LIN {X 0,Y 131.73,Z 570.995,A -85,B 0,C 180,E1 -25686.554,E2 -25686.554} C_VEL
LIN {X 0,Y 133.892,Z 570.97,A -85,B 0,C 180,E1 -25688.915,E2 -25688.915} C_VEL
LIN {X 0,Y 134.91,Z 571.003,A -85,B 0,C 180,E1 -25689.63,E2 -25689.63} C_VEL
LIN {X 0,Y 142.32,Z 571.103,A -85,B 0,C 180,E1 -25693.736,E2 -25693.736} C_VEL
LIN {X 0,Y 151.999,Z 570.353,A -85,B 0,C 180,E1 -25697.713,E2 -25697.713} C_VEL
LIN {X 0,Y 158.478,Z 569.41,A -85,B 0,C 180,E1 -25699.824,E2 -25699.824} C_VEL
LIN {X 0,Y 159.217,Z 569.07,A -85,B 0,C 180,E1 -25700.5,E2 -25700.5} C_VEL
LIN {X 0,Y 151.909,Z 567.926,A -85,B 0,C 180,E1 -25703.025,E2 -25703.025} C_VEL
LIN {X 0,Y 142.456,Z 565.139,A -85,B 0,C 180,E1 -25707.132,E2 -25707.132} C_VEL
LIN {X 0,Y 134.098,Z 561.047,A -85,B 0,C 180,E1 -25711.855,E2 -25711.855} C_VEL
LIN {X 0,Y 127.082,Z 555.595,A -85,B 0,C 180,E1 -25717.223,E2 -25717.223} C_VEL
LIN {X 0,Y 121.684,Z 548.605,A -85,B 0,C 180,E1 -25723.213,E2 -25723.213} C_VEL
LIN {X 0,Y 117.883,Z 539.949,A -85,B 0,C 180,E1 -25729.695,E2 -25729.695} C_VEL
LIN {X 0,Y 115.994,Z 530.669,A -85,B 0,C 180,E1 -25735.655,E2 -25735.655} C_VEL
LIN {X 0,Y 115.384,Z 519.452,A -85,B 0,C 180,E1 -25741.744,E2 -25741.744} C_VEL
LIN {X 0,Y 115.582,Z 508.598,A -85,B 0,C 180,E1 -25746.545,E2 -25746.545} C_VEL
LIN {X 0,Y 116.083,Z 497.899,A -85,B 0,C 180,E1 -25750.463,E2 -25750.463} C_VEL
LIN {X 0,Y 116.869,Z 485.455,A -85,B 0,C 180,E1 -25754.183,E2 -25754.183} C_VEL
LIN {X 0,Y 117.808,Z 470.89,A -85,B 0,C 180,E1 -25757.577,E2 -25757.577} C_VEL
LIN {X 0,Y 118.72,Z 456.9,A -85,B 0,C 180,E1 -25760.012,E2 -25760.012} C_VEL
LIN {X 0,Y 119.766,Z 433.179,A -85,B 0,C 180,E1 -25762.99,E2 -25762.99} C_VEL
LIN {X 0,Y 121.096,Z 391.719,A -85,B 0,C 180,E1 -25767.775,E2 -25767.775} C_VEL
LIN {X 0,Y 115.765,Z 370.385,A -85,B 0,C 180,E1 -25770.236,E2 -25770.236} C_VEL
LIN {X 0,Y 115.16,Z 367.133,A -85,B 0,C 180,E1 -25770.68,E2 -25770.68} C_VEL
LIN {X 0,Y 114.785,Z 367.181,A -85,B 0,C 180,E1 -25777.752,E2 -25777.752} C_VEL
LIN {X 0,Y 114.785,Z 367.188,A -85,B 0,C 180,E1 -25782.716,E2 -25782.716} C_VEL
LIN {X 0,Y 114.8,Z 367.179,A -85,B 0,C 180,E1 -25787.669,E2 -25787.669} C_VEL
LIN {X 0,Y 114.81,Z 367.183,A -85,B 0,C 180,E1 -25792.727,E2 -25792.727} C_VEL
LIN {X 0,Y 114.866,Z 367.177,A -85,B 0,C 180,E1 -25798.931,E2 -25798.931} C_VEL
LIN {X 0,Y 114.944,Z 367.165,A -85,B 0,C 180,E1 -25806.507,E2 -25806.507} C_VEL
LIN {X 0,Y 115.016,Z 367.152,A -85,B 0,C 180,E1 -25812.211,E2 -25812.211} C_VEL
LIN {X 0,Y 115.284,Z 367.124,A -85,B 0,C 180,E1 -25817.258,E2 -25817.258} C_VEL
LIN {X 0,Y 115.391,Z 367.108,A -85,B 0,C 180,E1 -25819.472,E2 -25819.472} C_VEL
LIN {X 0,Y 115.535,Z 367.093,A -85,B 0,C 180,E1 -25826.513,E2 -25826.513} C_VEL
LIN {X 0,Y 115.994,Z 367.029,A -85,B 0,C 180,E1 -25830.001,E2 -25830.001} C_VEL
LIN {X 0,Y 115.396,Z 367.106,A -85,B 0,C 180,E1 -25836.997,E2 -25836.997} C_VEL
LIN {X 0,Y 115.391,Z 367.109,A -85,B 0,C 180,E1 -25840.529,E2 -25840.529} C_VEL
LIN {X 0,Y 115.146,Z 367.141,A -85,B 0,C 180,E1 -25844.132,E2 -25844.132} C_VEL
LIN {X 0,Y 114.98,Z 367.162,A -85,B 0,C 180,E1 -25851.516,E2 -25851.516} C_VEL
LIN {X 0,Y 114.872,Z 367.169,A -85,B 0,C 180,E1 -25855.359,E2 -25855.359} C_VEL
LIN {X 0,Y 114.867,Z 367.175,A -85,B 0,C 180,E1 -25861.07,E2 -25861.07} C_VEL
LIN {X 0,Y 114.801,Z 367.185,A -85,B 0,C 180,E1 -25867.749,E2 -25867.749} C_VEL
LIN {X 0,Y 114.793,Z 367.179,A -85,B 0,C 180,E1 -25872.723,E2 -25872.723} C_VEL
LIN {X 0,Y 115,Z 367.154,A -85,B 0,C 180,E1 -25880.133,E2 -25880.133} C_VEL
LIN {X 0,Y 122.575,Z 395.545,A -85,B 0,C 180,E1 -25883.546,E2 -25883.546} C_VEL
LIN {X 0,Y 119.952,Z 450.842,A -85,B 0,C 180,E1 -25889.405,E2 -25889.405} C_VEL
LIN {X 0,Y 118.922,Z 465.573,A -85,B 0,C 180,E1 -25891.547,E2 -25891.547} C_VEL
LIN {X 0,Y 117.737,Z 479.37,A -85,B 0,C 180,E1 -25894.314,E2 -25894.314} C_VEL
LIN {X 0,Y 116.517,Z 492.918,A -85,B 0,C 180,E1 -25897.855,E2 -25897.855} C_VEL
LIN {X 0,Y 115.452,Z 506.149,A -85,B 0,C 180,E1 -25902.282,E2 -25902.282} C_VEL
LIN {X 0,Y 114.783,Z 517.895,A -85,B 0,C 180,E1 -25907.313,E2 -25907.313} C_VEL
LIN {X 0,Y 114.688,Z 527.291,A -85,B 0,C 180,E1 -25912.188,E2 -25912.188} C_VEL
LIN {X 0,Y 115.328,Z 535.667,A -85,B 0,C 180,E1 -25917.382,E2 -25917.382} C_VEL
LIN {X 0,Y 117.114,Z 543.83,A -85,B 0,C 180,E1 -25923.442,E2 -25923.442} C_VEL
LIN {X 0,Y 119.746,Z 549.675,A -85,B 0,C 180,E1 -25928.439,E2 -25928.439} C_VEL
LIN {X 0,Y 124.689,Z 555.877,A -85,B 0,C 180,E1 -25934.695,E2 -25934.695} C_VEL
LIN {X 0,Y 129.437,Z 559.537,A -85,B 0,C 180,E1 -25939.014,E2 -25939.014} C_VEL
LIN {X 0,Y 137.108,Z 563.055,A -85,B 0,C 180,E1 -25944.211,E2 -25944.211} C_VEL
LIN {X 0,Y 145.877,Z 565.201,A -85,B 0,C 180,E1 -25948.803,E2 -25948.803} C_VEL
LIN {X 0,Y 150.702,Z 565.75,A -85,B 0,C 180,E1 -25950.864,E2 -25950.864} C_VEL
LIN {X 0,Y 161.056,Z 565.721,A -85,B 0,C 180,E1 -25954.562,E2 -25954.562} C_VEL
LIN {X 0,Y 168.992,Z 564.854,A -85,B 0,C 180,E1 -25956.918,E2 -25956.918} C_VEL
LIN {X 0,Y 168.367,Z 565.266,A -85,B 0,C 180,E1 -25957.522,E2 -25957.522} C_VEL
LIN {X 0,Y 157.071,Z 568.845,A -85,B 0,C 180,E1 -25960.477,E2 -25960.477} C_VEL
LIN {X 0,Y 146.884,Z 571.301,A -85,B 0,C 180,E1 -25964.133,E2 -25964.133} C_VEL
LIN {X 0,Y 137.625,Z 572.661,A -85,B 0,C 180,E1 -25968.404,E2 -25968.404} C_VEL
LIN {X 0,Y 129.744,Z 572.964,A -85,B 0,C 180,E1 -25973.426,E2 -25973.426} C_VEL
LIN {X 0,Y 123.542,Z 572.25,A -85,B 0,C 180,E1 -25979.203,E2 -25979.203} C_VEL
LIN {X 0,Y 119.301,Z 570.519,A -85,B 0,C 180,E1 -25985.645,E2 -25985.645} C_VEL
LIN {X 0,Y 117.086,Z 567.075,A -85,B 0,C 180,E1 -25993.825,E2 -25993.825} C_VEL
LIN {X 0,Y 117.795,Z 562.438,A -85,B 0,C 180,E1 -26001.421,E2 -26001.421} C_VEL
LIN {X 0,Y 119.686,Z 558.145,A -85,B 0,C 180,E1 -26006.633,E2 -26006.633} C_VEL
LIN {X 0,Y 121.553,Z 553.452,A -85,B 0,C 180,E1 -26010.862,E2 -26010.862} C_VEL
LIN {X 0,Y 122.427,Z 551.524,A -85,B 0,C 180,E1 -26012.403,E2 -26012.403} C_VEL
LIN {X 0,Y 119.958,Z 557.118,A -85,B 0,C 180,E1 -26018.252,E2 -26018.252} C_VEL
LIN {X 0,Y 118.732,Z 562.143,A -85,B 0,C 180,E1 -26025.448,E2 -26025.448} C_VEL
LIN {X 0,Y 119.345,Z 565.021,A -85,B 0,C 180,E1 -26030.691,E2 -26030.691} C_VEL
LIN {X 0,Y 122.151,Z 567.945,A -85,B 0,C 180,E1 -26037.405,E2 -26037.405} C_VEL
LIN {X 0,Y 127.121,Z 569.905,A -85,B 0,C 180,E1 -26043.563,E2 -26043.563} C_VEL
LIN {X 0,Y 134.91,Z 571.003,A -85,B 0,C 180,E1 -26049.63,E2 -26049.63} C_VEL
LIN {X 0,Y 136.633,Z 570.98,A -85,B 0,C 180,E1 -26051.153,E2 -26051.153} C_VEL
LIN {X 0,Y 140.12,Z 569.71,A -85,B 0,C 180,E1 -26056.537,E2 -26056.537} C_VEL
LIN {X 0,Y 142.388,Z 569.441,A -85,B 0,C 180,E1 -26057.855,E2 -26057.855} C_VEL
LIN {X 0,Y 148.167,Z 569.104,A -85,B 0,C 180,E1 -26059.993,E2 -26059.993} C_VEL
LIN {X 0,Y 147.74,Z 568.702,A -85,B 0,C 180,E1 -26060.827,E2 -26060.827} C_VEL
LIN {X 0,Y 141.273,Z 566.851,A -85,B 0,C 180,E1 -26063.345,E2 -26063.345} C_VEL
LIN {X 0,Y 132.011,Z 562.872,A -85,B 0,C 180,E1 -26067.832,E2 -26067.832} C_VEL
LIN {X 0,Y 124.058,Z 557.572,A -85,B 0,C 180,E1 -26073.049,E2 -26073.049} C_VEL
LIN {X 0,Y 117.628,Z 550.855,A -85,B 0,C 180,E1 -26078.991,E2 -26078.991} C_VEL
LIN {X 0,Y 112.873,Z 542.487,A -85,B 0,C 180,E1 -26085.576,E2 -26085.576} C_VEL
LIN {X 0,Y 110.207,Z 533.661,A -85,B 0,C 180,E1 -26091.749,E2 -26091.749} C_VEL
LIN {X 0,Y 108.789,Z 522.89,A -85,B 0,C 180,E1 -26098.147,E2 -26098.147} C_VEL
LIN {X 0,Y 108.708,Z 512.813,A -85,B 0,C 180,E1 -26103.241,E2 -26103.241} C_VEL
LIN {X 0,Y 109.057,Z 501.757,A -85,B 0,C 180,E1 -26107.869,E2 -26107.869} C_VEL
LIN {X 0,Y 109.628,Z 489.445,A -85,B 0,C 180,E1 -26112.024,E2 -26112.024} C_VEL
LIN {X 0,Y 110.337,Z 478.245,A -85,B 0,C 180,E1 -26115.101,E2 -26115.101} C_VEL
LIN {X 0,Y 111.269,Z 464.295,A -85,B 0,C 180,E1 -26118.108,E2 -26118.108} C_VEL
LIN {X 0,Y 112.021,Z 449.968,A -85,B 0,C 180,E1 -26120.387,E2 -26120.387} C_VEL
LIN {X 0,Y 112.84,Z 428.51,A -85,B 0,C 180,E1 -26123.149,E2 -26123.149} C_VEL
LIN {X 0,Y 113.972,Z 392.449,A -85,B 0,C 180,E1 -26127.612,E2 -26127.612} C_VEL
LIN {X 0,Y 108.815,Z 371.696,A -85,B 0,C 180,E1 -26130.125,E2 -26130.125} C_VEL
LIN {X 0,Y 108.119,Z 368.01,A -85,B 0,C 180,E1 -26130.619,E2 -26130.619} C_VEL
LIN {X 0,Y 107.691,Z 368.063,A -85,B 0,C 180,E1 -26138.453,E2 -26138.453} C_VEL
LIN {X 0,Y 107.679,Z 368.068,A -85,B 0,C 180,E1 -26145.883,E2 -26145.883} C_VEL
LIN {X 0,Y 107.705,Z 368.068,A -85,B 0,C 180,E1 -26151.536,E2 -26151.536} C_VEL
LIN {X 0,Y 107.804,Z 368.055,A -85,B 0,C 180,E1 -26158.565,E2 -26158.565} C_VEL
LIN {X 0,Y 107.908,Z 368.043,A -85,B 0,C 180,E1 -26166.998,E2 -26166.998} C_VEL
LIN {X 0,Y 108.037,Z 368.026,A -85,B 0,C 180,E1 -26174.918,E2 -26174.918} C_VEL
LIN {X 0,Y 108.304,Z 367.992,A -85,B 0,C 180,E1 -26178.775,E2 -26178.775} C_VEL
LIN {X 0,Y 108.461,Z 367.975,A -85,B 0,C 180,E1 -26186.285,E2 -26186.285} C_VEL
LIN {X 0,Y 108.945,Z 367.907,A -85,B 0,C 180,E1 -26190.001,E2 -26190.001} C_VEL
LIN {X 0,Y 108.338,Z 367.985,A -85,B 0,C 180,E1 -26197.455,E2 -26197.455} C_VEL
LIN {X 0,Y 108.201,Z 368.007,A -85,B 0,C 180,E1 -26203.027,E2 -26203.027} C_VEL
LIN {X 0,Y 107.907,Z 368.042,A -85,B 0,C 180,E1 -26209.006,E2 -26209.006} C_VEL
LIN {X 0,Y 107.857,Z 368.045,A -85,B 0,C 180,E1 -26214.187,E2 -26214.187} C_VEL
LIN {X 0,Y 107.793,Z 368.055,A -85,B 0,C 180,E1 -26222.053,E2 -26222.053} C_VEL
LIN {X 0,Y 107.707,Z 368.069,A -85,B 0,C 180,E1 -26228.465,E2 -26228.465} C_VEL
LIN {X 0,Y 107.7,Z 368.069,A -85,B 0,C 180,E1 -26235.875,E2 -26235.875} C_VEL
LIN {X 0,Y 107.921,Z 368.037,A -85,B 0,C 180,E1 -26239.801,E2 -26239.801} C_VEL
LIN {X 0,Y 115.442,Z 397.023,A -85,B 0,C 180,E1 -26243.484,E2 -26243.484} C_VEL
LIN {X 0,Y 112.956,Z 448.955,A -85,B 0,C 180,E1 -26249.377,E2 -26249.377} C_VEL
LIN {X 0,Y 112.103,Z 462.355,A -85,B 0,C 180,E1 -26251.276,E2 -26251.276} C_VEL
LIN {X 0,Y 110.854,Z 476.95,A -85,B 0,C 180,E1 -26254.162,E2 -26254.162} C_VEL
LIN {X 0,Y 109.706,Z 489.289,A -85,B 0,C 180,E1 -26257.397,E2 -26257.397} C_VEL
LIN {X 0,Y 108.696,Z 502.041,A -85,B 0,C 180,E1 -26261.629,E2 -26261.629} C_VEL
LIN {X 0,Y 108.018,Z 513.424,A -85,B 0,C 180,E1 -26266.361,E2 -26266.361} C_VEL
LIN {X 0,Y 107.775,Z 524.013,A -85,B 0,C 180,E1 -26271.723,E2 -26271.723} C_VEL
LIN {X 0,Y 108.37,Z 532.92,A -85,B 0,C 180,E1 -26277.214,E2 -26277.214} C_VEL
LIN {X 0,Y 110.105,Z 541.774,A -85,B 0,C 180,E1 -26283.661,E2 -26283.661} C_VEL
LIN {X 0,Y 112.721,Z 548.038,A -85,B 0,C 180,E1 -26288.969,E2 -26288.969} C_VEL
LIN {X 0,Y 116.359,Z 553.32,A -85,B 0,C 180,E1 -26293.982,E2 -26293.982} C_VEL
LIN {X 0,Y 120.926,Z 557.672,A -85,B 0,C 180,E1 -26298.643,E2 -26298.643} C_VEL
LIN {X 0,Y 126.435,Z 561.187,A -85,B 0,C 180,E1 -26302.9,E2 -26302.9} C_VEL
LIN {X 0,Y 134.957,Z 564.601,A -85,B 0,C 180,E1 -26307.95,E2 -26307.95} C_VEL
LIN {X 0,Y 144.576,Z 566.649,A -85,B 0,C 180,E1 -26312.327,E2 -26312.327} C_VEL
LIN {X 0,Y 155.25,Z 567.233,A -85,B 0,C 180,E1 -26316.052,E2 -26316.052} C_VEL
LIN {X 0,Y 157.395,Z 567.196,A -85,B 0,C 180,E1 -26316.712,E2 -26316.712} C_VEL
LIN {X 0,Y 156.388,Z 567.621,A -85,B 0,C 180,E1 -26317.415,E2 -26317.415} C_VEL
LIN {X 0,Y 147.158,Z 569.663,A -85,B 0,C 180,E1 -26320.169,E2 -26320.169} C_VEL
LIN {X 0,Y 137.115,Z 571.121,A -85,B 0,C 180,E1 -26324.143,E2 -26324.143} C_VEL
LIN {X 0,Y 128.182,Z 571.545,A -85,B 0,C 180,E1 -26328.856,E2 -26328.856} C_VEL
LIN {X 0,Y 120.147,Z 570.844,A -85,B 0,C 180,E1 -26334.98,E2 -26334.98} C_VEL
LIN {X 0,Y 115.165,Z 569.388,A -85,B 0,C 180,E1 -26340.777,E2 -26340.777} C_VEL
LIN {X 0,Y 111.768,Z 566.813,A -85,B 0,C 180,E1 -26347.834,E2 -26347.834} C_VEL
LIN {X 0,Y 110.653,Z 563.069,A -85,B 0,C 180,E1 -26355.282,E2 -26355.282} C_VEL
LIN {X 0,Y 111.97,Z 558.027,A -85,B 0,C 180,E1 -26362.788,E2 -26362.788} C_VEL
LIN {X 0,Y 113.82,Z 553.912,A -85,B 0,C 180,E1 -26367.505,E2 -26367.505} C_VEL
LIN {X 0,Y 116.373,Z 547.902,A -85,B 0,C 180,E1 -26372.704,E2 -26372.704} C_VEL
LIN {X 0,Y 114.439,Z 552.194,A -85,B 0,C 180,E1 -26377.055,E2 -26377.055} C_VEL
LIN {X 0,Y 112.69,Z 557.762,A -85,B 0,C 180,E1 -26384.445,E2 -26384.445} C_VEL
LIN {X 0,Y 113.31,Z 562.033,A -85,B 0,C 180,E1 -26391.848,E2 -26391.848} C_VEL
LIN {X 0,Y 116.311,Z 565.247,A -85,B 0,C 180,E1 -26398.907,E2 -26398.907} C_VEL
LIN {X 0,Y 121.576,Z 567.556,A -85,B 0,C 180,E1 -26405.315,E2 -26405.315} C_VEL
LIN {X 0,Y 129.378,Z 569.016,A -85,B 0,C 180,E1 -26411.353,E2 -26411.353} C_VEL
LIN {X 0,Y 137.411,Z 569.493,A -85,B 0,C 180,E1 -26415.728,E2 -26415.728} C_VEL
LIN {X 0,Y 142.388,Z 569.441,A -85,B 0,C 180,E1 -26417.855,E2 -26417.855} C_VEL
LIN {X 0,Y 142.985,Z 569.237,A -85,B 0,C 180,E1 -26418.515,E2 -26418.515} C_VEL
LIN {X 0,Y 142.417,Z 568.762,A -85,B 0,C 180,E1 -26419.453,E2 -26419.453} C_VEL
LIN {X 0,Y 140.261,Z 567.932,A -85,B 0,C 180,E1 -26420.671,E2 -26420.671} C_VEL
LIN {X 0,Y 130.281,Z 564.415,A -85,B 0,C 180,E1 -26423.995,E2 -26423.995} C_VEL
LIN {X 0,Y 129.151,Z 563.873,A -85,B 0,C 180,E1 -26424.505,E2 -26424.505} C_VEL
LIN {X 0,Y 121.769,Z 559.467,A -85,B 0,C 180,E1 -26428.703,E2 -26428.703} C_VEL
LIN {X 0,Y 114.249,Z 552.922,A -85,B 0,C 180,E1 -26434.492,E2 -26434.492} C_VEL
LIN {X 0,Y 108.469,Z 544.852,A -85,B 0,C 180,E1 -26441.095,E2 -26441.095} C_VEL
LIN {X 0,Y 104.506,Z 535.008,A -85,B 0,C 180,E1 -26448.359,E2 -26448.359} C_VEL
LIN {X 0,Y 102.697,Z 526.105,A -85,B 0,C 180,E1 -26454.106,E2 -26454.106} C_VEL
LIN {X 0,Y 102.129,Z 515.639,A -85,B 0,C 180,E1 -26459.998,E2 -26459.998} C_VEL
LIN {X 0,Y 102.206,Z 503.981,A -85,B 0,C 180,E1 -26465.423,E2 -26465.423} C_VEL
LIN {X 0,Y 102.645,Z 492.254,A -85,B 0,C 180,E1 -26469.854,E2 -26469.854} C_VEL
LIN {X 0,Y 103.395,Z 479.347,A -85,B 0,C 180,E1 -26473.761,E2 -26473.761} C_VEL
LIN {X 0,Y 104.245,Z 465.456,A -85,B 0,C 180,E1 -26477.021,E2 -26477.021} C_VEL
LIN {X 0,Y 104.986,Z 451.448,A -85,B 0,C 180,E1 -26479.46,E2 -26479.46} C_VEL
LIN {X 0,Y 105.828,Z 428.168,A -85,B 0,C 180,E1 -26482.698,E2 -26482.698} C_VEL
LIN {X 0,Y 106.872,Z 393.068,A -85,B 0,C 180,E1 -26487.39,E2 -26487.39} C_VEL
LIN {X 0,Y 102.002,Z 373.826,A -85,B 0,C 180,E1 -26489.829,E2 -26489.829} C_VEL
LIN {X 0,Y 101.057,Z 368.889,A -85,B 0,C 180,E1 -26490.576,E2 -26490.576} C_VEL
LIN {X 0,Y 100.641,Z 368.944,A -85,B 0,C 180,E1 -26499.812,E2 -26499.812} C_VEL
LIN {X 0,Y 100.649,Z 368.943,A -85,B 0,C 180,E1 -26505.713,E2 -26505.713} C_VEL
LIN {X 0,Y 100.643,Z 368.949,A -85,B 0,C 180,E1 -26511.063,E2 -26511.063} C_VEL
LIN {X 0,Y 100.697,Z 368.936,A -85,B 0,C 180,E1 -26516.876,E2 -26516.876} C_VEL
LIN {X 0,Y 100.783,Z 368.926,A -85,B 0,C 180,E1 -26525.267,E2 -26525.267} C_VEL
LIN {X 0,Y 100.816,Z 368.926,A -85,B 0,C 180,E1 -26529.602,E2 -26529.602} C_VEL
LIN {X 0,Y 101.197,Z 368.879,A -85,B 0,C 180,E1 -26537.975,E2 -26537.975} C_VEL
LIN {X 0,Y 101.277,Z 368.862,A -85,B 0,C 180,E1 -26542.023,E2 -26542.023} C_VEL
LIN {X 0,Y 101.869,Z 368.788,A -85,B 0,C 180,E1 -26550.001,E2 -26550.001} C_VEL
LIN {X 0,Y 101.277,Z 368.862,A -85,B 0,C 180,E1 -26557.978,E2 -26557.978} C_VEL
LIN {X 0,Y 101.127,Z 368.888,A -85,B 0,C 180,E1 -26563.364,E2 -26563.364} C_VEL
LIN {X 0,Y 100.817,Z 368.927,A -85,B 0,C 180,E1 -26570.4,E2 -26570.4} C_VEL
LIN {X 0,Y 100.772,Z 368.925,A -85,B 0,C 180,E1 -26574.96,E2 -26574.96} C_VEL
LIN {X 0,Y 100.699,Z 368.936,A -85,B 0,C 180,E1 -26583.126,E2 -26583.126} C_VEL
LIN {X 0,Y 100.653,Z 368.946,A -85,B 0,C 180,E1 -26589.823,E2 -26589.823} C_VEL
LIN {X 0,Y 100.735,Z 368.937,A -85,B 0,C 180,E1 -26597.677,E2 -26597.677} C_VEL
LIN {X 0,Y 100.856,Z 368.919,A -85,B 0,C 180,E1 -26599.422,E2 -26599.422} C_VEL
LIN {X 0,Y 108.313,Z 397.297,A -85,B 0,C 180,E1 -26603.322,E2 -26603.322} C_VEL
LIN {X 0,Y 105.803,Z 450.176,A -85,B 0,C 180,E1 -26609.764,E2 -26609.764} C_VEL
LIN {X 0,Y 104.804,Z 464.348,A -85,B 0,C 180,E1 -26612.006,E2 -26612.006} C_VEL
LIN {X 0,Y 103.691,Z 477.843,A -85,B 0,C 180,E1 -26614.939,E2 -26614.939} C_VEL
LIN {X 0,Y 102.501,Z 491.663,A -85,B 0,C 180,E1 -26618.904,E2 -26618.904} C_VEL
LIN {X 0,Y 101.56,Z 504.019,A -85,B 0,C 180,E1 -26623.416,E2 -26623.416} C_VEL
LIN {X 0,Y 101.056,Z 515.189,A -85,B 0,C 180,E1 -26628.524,E2 -26628.524} C_VEL
LIN {X 0,Y 101.076,Z 525.08,A -85,B 0,C 180,E1 -26634.015,E2 -26634.015} C_VEL
LIN {X 0,Y 101.968,Z 534.167,A -85,B 0,C 180,E1 -26640.002,E2 -26640.002} C_VEL
LIN {X 0,Y 104.308,Z 542.865,A -85,B 0,C 180,E1 -26646.773,E2 -26646.773} C_VEL
LIN {X 0,Y 108.45,Z 550.55,A -85,B 0,C 180,E1 -26653.571,E2 -26653.571} C_VEL
LIN {X 0,Y 114.153,Z 556.667,A -85,B 0,C 180,E1 -26659.794,E2 -26659.794} C_VEL
LIN {X 0,Y 121.927,Z 561.786,A -85,B 0,C 180,E1 -26665.616,E2 -26665.616} C_VEL
LIN {X 0,Y 130.205,Z 565.199,A -85,B 0,C 180,E1 -26670.273,E2 -26670.273} C_VEL
LIN {X 0,Y 138.53,Z 567.276,A -85,B 0,C 180,E1 -26673.923,E2 -26673.923} C_VEL
LIN {X 0,Y 145.297,Z 568.179,A -85,B 0,C 180,E1 -26676.336,E2 -26676.336} C_VEL
LIN {X 0,Y 145.337,Z 568.514,A -85,B 0,C 180,E1 -26677.181,E2 -26677.181} C_VEL
LIN {X 0,Y 137.441,Z 569.564,A -85,B 0,C 180,E1 -26679.912,E2 -26679.912} C_VEL
LIN {X 0,Y 127.532,Z 570.065,A -85,B 0,C 180,E1 -26684.241,E2 -26684.241} C_VEL
LIN {X 0,Y 118.921,Z 569.589,A -85,B 0,C 180,E1 -26689.452,E2 -26689.452} C_VEL
LIN {X 0,Y 112.027,Z 568.154,A -85,B 0,C 180,E1 -26695.624,E2 -26695.624} C_VEL
LIN {X 0,Y 107.17,Z 565.742,A -85,B 0,C 180,E1 -26702.674,E2 -26702.674} C_VEL
LIN {X 0,Y 104.68,Z 562.305,A -85,B 0,C 180,E1 -26710.385,E2 -26710.385} C_VEL
LIN {X 0,Y 104.698,Z 557.655,A -85,B 0,C 180,E1 -26718.382,E2 -26718.382} C_VEL
LIN {X 0,Y 106.611,Z 552.655,A -85,B 0,C 180,E1 -26724.969,E2 -26724.969} C_VEL
LIN {X 0,Y 108.212,Z 549.042,A -85,B 0,C 180,E1 -26728.688,E2 -26728.688} C_VEL
LIN {X 0,Y 110.431,Z 544.057,A -85,B 0,C 180,E1 -26732.963,E2 -26732.963} C_VEL
LIN {X 0,Y 107.831,Z 550.004,A -85,B 0,C 180,E1 -26739.347,E2 -26739.347} C_VEL
LIN {X 0,Y 106.643,Z 555.518,A -85,B 0,C 180,E1 -26747.251,E2 -26747.251} C_VEL
LIN {X 0,Y 107.682,Z 559.298,A -85,B 0,C 180,E1 -26753.97,E2 -26753.97} C_VEL
LIN {X 0,Y 110.644,Z 562.372,A -85,B 0,C 180,E1 -26760.54,E2 -26760.54} C_VEL
LIN {X 0,Y 116.209,Z 564.999,A -85,B 0,C 180,E1 -26767.212,E2 -26767.212} C_VEL
LIN {X 0,Y 123.685,Z 566.754,A -85,B 0,C 180,E1 -26772.989,E2 -26772.989} C_VEL
LIN {X 0,Y 132.707,Z 567.665,A -85,B 0,C 180,E1 -26777.853,E2 -26777.853} C_VEL
LIN {X 0,Y 137.74,Z 567.829,A -85,B 0,C 180,E1 -26779.938,E2 -26779.938} C_VEL
LIN {X 0,Y 135.619,Z 566.74,A -85,B 0,C 180,E1 -26781.546,E2 -26781.546} C_VEL
LIN {X 0,Y 129.151,Z 563.873,A -85,B 0,C 180,E1 -26784.505,E2 -26784.505} C_VEL
LIN {X 0,Y 125.052,Z 561.898,A -85,B 0,C 180,E1 -26786.194,E2 -26786.194} C_VEL
LIN {X 0,Y 117.535,Z 557.99,A -85,B 0,C 180,E1 -26788.616,E2 -26788.616} C_VEL
LIN {X 0,Y 110.563,Z 553.432,A -85,B 0,C 180,E1 -26791.319,E2 -26791.319} C_VEL
LIN {X 0,Y 107.432,Z 550.487,A -85,B 0,C 180,E1 -26793.466,E2 -26793.466} C_VEL
LIN {X 0,Y 102.048,Z 542.527,A -85,B 0,C 180,E1 -26799.856,E2 -26799.856} C_VEL
LIN {X 0,Y 98.349,Z 533.439,A -85,B 0,C 180,E1 -26806.569,E2 -26806.569} C_VEL
LIN {X 0,Y 96.333,Z 524.228,A -85,B 0,C 180,E1 -26812.663,E2 -26812.663} C_VEL
LIN {X 0,Y 95.624,Z 512.433,A -85,B 0,C 180,E1 -26819.472,E2 -26819.472} C_VEL
LIN {X 0,Y 95.671,Z 500.014,A -85,B 0,C 180,E1 -26825.267,E2 -26825.267} C_VEL
LIN {X 0,Y 95.984,Z 488.855,A -85,B 0,C 180,E1 -26829.48,E2 -26829.48} C_VEL
LIN {X 0,Y 96.652,Z 476.969,A -85,B 0,C 180,E1 -26833.132,E2 -26833.132} C_VEL
LIN {X 0,Y 97.467,Z 463.014,A -85,B 0,C 180,E1 -26836.492,E2 -26836.492} C_VEL
LIN {X 0,Y 98.225,Z 447.286,A -85,B 0,C 180,E1 -26839.197,E2 -26839.197} C_VEL
LIN {X 0,Y 98.839,Z 425.783,A -85,B 0,C 180,E1 -26842.427,E2 -26842.427} C_VEL
LIN {X 0,Y 99.795,Z 393.897,A -85,B 0,C 180,E1 -26847.043,E2 -26847.043} C_VEL
LIN {X 0,Y 95.075,Z 375.23,A -85,B 0,C 180,E1 -26849.538,E2 -26849.538} C_VEL
LIN {X 0,Y 94.03,Z 369.764,A -85,B 0,C 180,E1 -26850.405,E2 -26850.405} C_VEL
LIN {X 0,Y 93.549,Z 369.827,A -85,B 0,C 180,E1 -26856.939,E2 -26856.939} C_VEL
LIN {X 0,Y 93.533,Z 369.834,A -85,B 0,C 180,E1 -26862.549,E2 -26862.549} C_VEL
LIN {X 0,Y 93.542,Z 369.828,A -85,B 0,C 180,E1 -26868.702,E2 -26868.702} C_VEL
LIN {X 0,Y 93.595,Z 369.818,A -85,B 0,C 180,E1 -26875.684,E2 -26875.684} C_VEL
LIN {X 0,Y 93.666,Z 369.81,A -85,B 0,C 180,E1 -26884.204,E2 -26884.204} C_VEL
LIN {X 0,Y 93.692,Z 369.814,A -85,B 0,C 180,E1 -26887.973,E2 -26887.973} C_VEL
LIN {X 0,Y 94.095,Z 369.764,A -85,B 0,C 180,E1 -26897.052,E2 -26897.052} C_VEL
LIN {X 0,Y 94.209,Z 369.741,A -85,B 0,C 180,E1 -26901.42,E2 -26901.42} C_VEL
LIN {X 0,Y 94.796,Z 369.669,A -85,B 0,C 180,E1 -26910.001,E2 -26910.001} C_VEL
LIN {X 0,Y 94.209,Z 369.742,A -85,B 0,C 180,E1 -26918.581,E2 -26918.581} C_VEL
LIN {X 0,Y 94.045,Z 369.77,A -85,B 0,C 180,E1 -26923.723,E2 -26923.723} C_VEL
LIN {X 0,Y 93.693,Z 369.815,A -85,B 0,C 180,E1 -26932.029,E2 -26932.029} C_VEL
LIN {X 0,Y 93.622,Z 369.818,A -85,B 0,C 180,E1 -26936.771,E2 -26936.771} C_VEL
LIN {X 0,Y 93.597,Z 369.819,A -85,B 0,C 180,E1 -26944.317,E2 -26944.317} C_VEL
LIN {X 0,Y 93.544,Z 369.825,A -85,B 0,C 180,E1 -26952.547,E2 -26952.547} C_VEL
LIN {X 0,Y 93.808,Z 369.947,A -85,B 0,C 180,E1 -26959.235,E2 -26959.235} C_VEL
LIN {X 0,Y 101.165,Z 398.825,A -85,B 0,C 180,E1 -26963.341,E2 -26963.341} C_VEL
LIN {X 0,Y 98.746,Z 449.939,A -85,B 0,C 180,E1 -26970.121,E2 -26970.121} C_VEL
LIN {X 0,Y 97.772,Z 463.991,A -85,B 0,C 180,E1 -26972.438,E2 -26972.438} C_VEL
LIN {X 0,Y 96.629,Z 477.613,A -85,B 0,C 180,E1 -26975.567,E2 -26975.567} C_VEL
LIN {X 0,Y 95.533,Z 490.843,A -85,B 0,C 180,E1 -26979.549,E2 -26979.549} C_VEL
LIN {X 0,Y 94.67,Z 503.255,A -85,B 0,C 180,E1 -26984.373,E2 -26984.373} C_VEL
LIN {X 0,Y 94.26,Z 513.764,A -85,B 0,C 180,E1 -26989.39,E2 -26989.39} C_VEL
LIN {X 0,Y 94.434,Z 524.703,A -85,B 0,C 180,E1 -26995.734,E2 -26995.734} C_VEL
LIN {X 0,Y 95.617,Z 533.87,A -85,B 0,C 180,E1 -27002.108,E2 -27002.108} C_VEL
LIN {X 0,Y 98.309,Z 542.771,A -85,B 0,C 180,E1 -27009.258,E2 -27009.258} C_VEL
LIN {X 0,Y 102.668,Z 550.113,A -85,B 0,C 180,E1 -27015.893,E2 -27015.893} C_VEL
LIN {X 0,Y 109.318,Z 556.975,A -85,B 0,C 180,E1 -27022.691,E2 -27022.691} C_VEL
LIN {X 0,Y 117.714,Z 562.26,A -85,B 0,C 180,E1 -27028.533,E2 -27028.533} C_VEL
LIN {X 0,Y 127.352,Z 566.167,A -85,B 0,C 180,E1 -27033.496,E2 -27033.496} C_VEL
LIN {X 0,Y 134.813,Z 568.086,A -85,B 0,C 180,E1 -27036.496,E2 -27036.496} C_VEL
LIN {X 0,Y 134.106,Z 568.321,A -85,B 0,C 180,E1 -27037.218,E2 -27037.218} C_VEL
LIN {X 0,Y 122.798,Z 568.472,A -85,B 0,C 180,E1 -27041.924,E2 -27041.924} C_VEL
LIN {X 0,Y 113.82,Z 567.609,A -85,B 0,C 180,E1 -27047.217,E2 -27047.217} C_VEL
LIN {X 0,Y 106.538,Z 565.836,A -85,B 0,C 180,E1 -27053.579,E2 -27053.579} C_VEL
LIN {X 0,Y 101.323,Z 563.112,A -85,B 0,C 180,E1 -27060.952,E2 -27060.952} C_VEL
LIN {X 0,Y 98.306,Z 558.222,A -85,B 0,C 180,E1 -27071.233,E2 -27071.233} C_VEL
LIN {X 0,Y 98.969,Z 552.758,A -85,B 0,C 180,E1 -27079.98,E2 -27079.98} C_VEL
LIN {X 0,Y 101.037,Z 547.937,A -85,B 0,C 180,E1 -27086.011,E2 -27086.011} C_VEL
LIN {X 0,Y 104.613,Z 540.036,A -85,B 0,C 180,E1 -27093.249,E2 -27093.249} C_VEL
LIN {X 0,Y 102.199,Z 545.513,A -85,B 0,C 180,E1 -27099.123,E2 -27099.123} C_VEL
LIN {X 0,Y 100.8,Z 551.928,A -85,B 0,C 180,E1 -27108.285,E2 -27108.285} C_VEL
LIN {X 0,Y 102.505,Z 556.753,A -85,B 0,C 180,E1 -27116.957,E2 -27116.957} C_VEL
LIN {X 0,Y 107.818,Z 560.868,A -85,B 0,C 180,E1 -27125.919,E2 -27125.919} C_VEL
LIN {X 0,Y 116.51,Z 563.834,A -85,B 0,C 180,E1 -27133.624,E2 -27133.624} C_VEL
LIN {X 0,Y 128.245,Z 565.622,A -85,B 0,C 180,E1 -27140.104,E2 -27140.104} C_VEL
LIN {X 0,Y 124.098,Z 563.469,A -85,B 0,C 180,E1 -27142.269,E2 -27142.269} C_VEL
LIN {X 0,Y 115.811,Z 558.255,A -85,B 0,C 180,E1 -27146.894,E2 -27146.894} C_VEL
LIN {X 0,Y 107.432,Z 550.487,A -85,B 0,C 180,E1 -27153.466,E2 -27153.466} C_VEL
LIN {X 0,Y 104.571,Z 547.384,A -85,B 0,C 180,E1 -27155.69,E2 -27155.69} C_VEL
LIN {X 0,Y 98.992,Z 541.544,A -85,B 0,C 180,E1 -27158.914,E2 -27158.914} C_VEL
LIN {X 0,Y 94.01,Z 535.143,A -85,B 0,C 180,E1 -27162.349,E2 -27162.349} C_VEL
LIN {X 0,Y 92.213,Z 531.224,A -85,B 0,C 180,E1 -27164.878,E2 -27164.878} C_VEL
LIN {X 0,Y 89.85,Z 520.379,A -85,B 0,C 180,E1 -27172.13,E2 -27172.13} C_VEL
LIN {X 0,Y 89.217,Z 509.893,A -85,B 0,C 180,E1 -27178.305,E2 -27178.305} C_VEL
LIN {X 0,Y 89.17,Z 496.905,A -85,B 0,C 180,E1 -27184.518,E2 -27184.518} C_VEL
LIN {X 0,Y 89.557,Z 483.407,A -85,B 0,C 180,E1 -27189.597,E2 -27189.597} C_VEL
LIN {X 0,Y 90.165,Z 470.11,A -85,B 0,C 180,E1 -27193.521,E2 -27193.521} C_VEL
LIN {X 0,Y 90.959,Z 456.472,A -85,B 0,C 180,E1 -27196.552,E2 -27196.552} C_VEL
LIN {X 0,Y 91.763,Z 432.527,A -85,B 0,C 180,E1 -27200.597,E2 -27200.597} C_VEL
LIN {X 0,Y 92.621,Z 394.364,A -85,B 0,C 180,E1 -27206.612,E2 -27206.612} C_VEL
LIN {X 0,Y 87.975,Z 375.646,A -85,B 0,C 180,E1 -27209.29,E2 -27209.29} C_VEL
LIN {X 0,Y 87.017,Z 370.637,A -85,B 0,C 180,E1 -27210.117,E2 -27210.117} C_VEL
LIN {X 0,Y 86.461,Z 370.712,A -85,B 0,C 180,E1 -27220.56,E2 -27220.56} C_VEL
LIN {X 0,Y 86.478,Z 370.705,A -85,B 0,C 180,E1 -27227.002,E2 -27227.002} C_VEL
LIN {X 0,Y 86.54,Z 370.696,A -85,B 0,C 180,E1 -27235.356,E2 -27235.356} C_VEL
LIN {X 0,Y 86.582,Z 370.693,A -85,B 0,C 180,E1 -27243.233,E2 -27243.233} C_VEL
LIN {X 0,Y 86.661,Z 370.686,A -85,B 0,C 180,E1 -27251.072,E2 -27251.072} C_VEL
LIN {X 0,Y 86.967,Z 370.651,A -85,B 0,C 180,E1 -27255.97,E2 -27255.97} C_VEL
LIN {X 0,Y 87.115,Z 370.625,A -85,B 0,C 180,E1 -27260.716,E2 -27260.716} C_VEL
LIN {X 0,Y 87.723,Z 370.55,A -85,B 0,C 180,E1 -27270.001,E2 -27270.001} C_VEL
LIN {X 0,Y 87.116,Z 370.627,A -85,B 0,C 180,E1 -27279.286,E2 -27279.286} C_VEL
LIN {X 0,Y 86.948,Z 370.653,A -85,B 0,C 180,E1 -27284.089,E2 -27284.089} C_VEL
LIN {X 0,Y 86.662,Z 370.687,A -85,B 0,C 180,E1 -27288.929,E2 -27288.929} C_VEL
LIN {X 0,Y 86.584,Z 370.694,A -85,B 0,C 180,E1 -27296.769,E2 -27296.769} C_VEL
LIN {X 0,Y 86.516,Z 370.703,A -85,B 0,C 180,E1 -27305.679,E2 -27305.679} C_VEL
LIN {X 0,Y 86.494,Z 370.703,A -85,B 0,C 180,E1 -27313.009,E2 -27313.009} C_VEL
LIN {X 0,Y 86.744,Z 370.883,A -85,B 0,C 180,E1 -27318.938,E2 -27318.938} C_VEL
LIN {X 0,Y 94.059,Z 399.18,A -85,B 0,C 180,E1 -27323.293,E2 -27323.293} C_VEL
LIN {X 0,Y 91.667,Z 450.029,A -85,B 0,C 180,E1 -27330.586,E2 -27330.586} C_VEL
LIN {X 0,Y 90.636,Z 464.737,A -85,B 0,C 180,E1 -27333.214,E2 -27333.214} C_VEL
LIN {X 0,Y 89.635,Z 477.151,A -85,B 0,C 180,E1 -27336.309,E2 -27336.309} C_VEL
LIN {X 0,Y 88.666,Z 489.672,A -85,B 0,C 180,E1 -27340.316,E2 -27340.316} C_VEL
LIN {X 0,Y 87.831,Z 502.71,A -85,B 0,C 180,E1 -27345.65,E2 -27345.65} C_VEL
LIN {X 0,Y 87.537,Z 513.897,A -85,B 0,C 180,E1 -27351.344,E2 -27351.344} C_VEL
LIN {X 0,Y 87.955,Z 524.118,A -85,B 0,C 180,E1 -27357.712,E2 -27357.712} C_VEL
LIN {X 0,Y 89.354,Z 533.444,A -85,B 0,C 180,E1 -27364.513,E2 -27364.513} C_VEL
LIN {X 0,Y 92.576,Z 542.511,A -85,B 0,C 180,E1 -27372.052,E2 -27372.052} C_VEL
LIN {X 0,Y 97.467,Z 550.094,A -85,B 0,C 180,E1 -27378.936,E2 -27378.936} C_VEL
LIN {X 0,Y 104.783,Z 557.098,A -85,B 0,C 180,E1 -27385.849,E2 -27385.849} C_VEL
LIN {X 0,Y 113.821,Z 562.691,A -85,B 0,C 180,E1 -27391.66,E2 -27391.66} C_VEL
LIN {X 0,Y 121.385,Z 565.913,A -85,B 0,C 180,E1 -27395.381,E2 -27395.381} C_VEL
LIN {X 0,Y 123.495,Z 566.983,A -85,B 0,C 180,E1 -27397.18,E2 -27397.18} C_VEL
LIN {X 0,Y 113.435,Z 566.184,A -85,B 0,C 180,E1 -27401.971,E2 -27401.971} C_VEL
LIN {X 0,Y 104.855,Z 564.506,A -85,B 0,C 180,E1 -27407.912,E2 -27407.912} C_VEL
LIN {X 0,Y 98.163,Z 561.924,A -85,B 0,C 180,E1 -27415.056,E2 -27415.056} C_VEL
LIN {X 0,Y 93.395,Z 557.782,A -85,B 0,C 180,E1 -27424.56,E2 -27424.56} C_VEL
LIN {X 0,Y 92.215,Z 552.411,A -85,B 0,C 180,E1 -27434.528,E2 -27434.528} C_VEL
LIN {X 0,Y 94.354,Z 545.666,A -85,B 0,C 180,E1 -27444.045,E2 -27444.045} C_VEL
LIN {X 0,Y 96.315,Z 540.96,A -85,B 0,C 180,E1 -27448.954,E2 -27448.954} C_VEL
LIN {X 0,Y 98.963,Z 535.759,A -85,B 0,C 180,E1 -27453.499,E2 -27453.499} C_VEL
LIN {X 0,Y 96.5,Z 541.413,A -85,B 0,C 180,E1 -27459.667,E2 -27459.667} C_VEL
LIN {X 0,Y 95.091,Z 548.16,A -85,B 0,C 180,E1 -27469.425,E2 -27469.425} C_VEL
LIN {X 0,Y 97.014,Z 553.27,A -85,B 0,C 180,E1 -27478.619,E2 -27478.619} C_VEL
LIN {X 0,Y 102.706,Z 557.738,A -85,B 0,C 180,E1 -27488.014,E2 -27488.014} C_VEL
LIN {X 0,Y 109.995,Z 560.592,A -85,B 0,C 180,E1 -27494.654,E2 -27494.654} C_VEL
LIN {X 0,Y 117.561,Z 562.381,A -85,B 0,C 180,E1 -27499.353,E2 -27499.353} C_VEL
LIN {X 0,Y 118.484,Z 562.405,A -85,B 0,C 180,E1 -27500.197,E2 -27500.197} C_VEL
LIN {X 0,Y 109.997,Z 556.731,A -85,B 0,C 180,E1 -27504.896,E2 -27504.896} C_VEL
LIN {X 0,Y 101.858,Z 548.99,A -85,B 0,C 180,E1 -27511.214,E2 -27511.214} C_VEL
LIN {X 0,Y 96.399,Z 541.129,A -85,B 0,C 180,E1 -27517.494,E2 -27517.494} C_VEL
LIN {X 0,Y 92.213,Z 531.224,A -85,B 0,C 180,E1 -27524.878,E2 -27524.878} C_VEL
LIN {X 0,Y 90.703,Z 527.28,A -85,B 0,C 180,E1 -27527.381,E2 -27527.381} C_VEL
LIN {X 0,Y 87.135,Z 519.992,A -85,B 0,C 180,E1 -27530.927,E2 -27530.927} C_VEL
LIN {X 0,Y 84.387,Z 513.643,A -85,B 0,C 180,E1 -27533.705,E2 -27533.705} C_VEL
LIN {X 0,Y 83.114,Z 508.815,A -85,B 0,C 180,E1 -27536.024,E2 -27536.024} C_VEL
LIN {X 0,Y 82.94,Z 507.215,A -85,B 0,C 180,E1 -27536.875,E2 -27536.875} C_VEL
LIN {X 0,Y 82.749,Z 496.179,A -85,B 0,C 180,E1 -27542.432,E2 -27542.432} C_VEL
LIN {X 0,Y 82.96,Z 482.531,A -85,B 0,C 180,E1 -27547.91,E2 -27547.91} C_VEL
LIN {X 0,Y 83.459,Z 470.12,A -85,B 0,C 180,E1 -27551.842,E2 -27551.842} C_VEL
LIN {X 0,Y 84.224,Z 454.99,A -85,B 0,C 180,E1 -27555.423,E2 -27555.423} C_VEL
LIN {X 0,Y 84.871,Z 429.283,A -85,B 0,C 180,E1 -27560.129,E2 -27560.129} C_VEL
LIN {X 0,Y 85.564,Z 395.153,A -85,B 0,C 180,E1 -27565.994,E2 -27565.994} C_VEL
LIN {X 0,Y 80.899,Z 376.159,A -85,B 0,C 180,E1 -27568.892,E2 -27568.892} C_VEL
LIN {X 0,Y 80,Z 371.511,A -85,B 0,C 180,E1 -27569.684,E2 -27569.684} C_VEL
LIN {X 0,Y 79.384,Z 371.588,A -85,B 0,C 180,E1 -27578.293,E2 -27578.293} C_VEL
LIN {X 0,Y 79.407,Z 371.59,A -85,B 0,C 180,E1 -27585.073,E2 -27585.073} C_VEL
LIN {X 0,Y 79.391,Z 371.594,A -85,B 0,C 180,E1 -27592.814,E2 -27592.814} C_VEL
LIN {X 0,Y 79.382,Z 371.594,A -85,B 0,C 180,E1 -27597.914,E2 -27597.914} C_VEL
LIN {X 0,Y 79.523,Z 371.571,A -85,B 0,C 180,E1 -27603.777,E2 -27603.777} C_VEL
LIN {X 0,Y 79.521,Z 371.579,A -85,B 0,C 180,E1 -27609.298,E2 -27609.298} C_VEL
LIN {X 0,Y 79.839,Z 371.539,A -85,B 0,C 180,E1 -27615.525,E2 -27615.525} C_VEL
LIN {X 0,Y 79.998,Z 371.514,A -85,B 0,C 180,E1 -27619.881,E2 -27619.881} C_VEL
LIN {X 0,Y 80.651,Z 371.43,A -85,B 0,C 180,E1 -27630.001,E2 -27630.001} C_VEL
LIN {X 0,Y 79.998,Z 371.515,A -85,B 0,C 180,E1 -27640.121,E2 -27640.121} C_VEL
LIN {X 0,Y 79.763,Z 371.545,A -85,B 0,C 180,E1 -27645.328,E2 -27645.328} C_VEL
LIN {X 0,Y 79.522,Z 371.58,A -85,B 0,C 180,E1 -27650.703,E2 -27650.703} C_VEL
LIN {X 0,Y 79.482,Z 371.582,A -85,B 0,C 180,E1 -27657.849,E2 -27657.849} C_VEL
LIN {X 0,Y 79.383,Z 371.593,A -85,B 0,C 180,E1 -27662.088,E2 -27662.088} C_VEL
LIN {X 0,Y 79.372,Z 371.599,A -85,B 0,C 180,E1 -27668.304,E2 -27668.304} C_VEL
LIN {X 0,Y 79.675,Z 371.558,A -85,B 0,C 180,E1 -27678.572,E2 -27678.572} C_VEL
LIN {X 0,Y 85.855,Z 395.917,A -85,B 0,C 180,E1 -27682.705,E2 -27682.705} C_VEL
LIN {X 0,Y 86.882,Z 400.375,A -85,B 0,C 180,E1 -27683.382,E2 -27683.382} C_VEL
LIN {X 0,Y 84.597,Z 450.368,A -85,B 0,C 180,E1 -27691.299,E2 -27691.299} C_VEL
LIN {X 0,Y 83.589,Z 464.984,A -85,B 0,C 180,E1 -27694.144,E2 -27694.144} C_VEL
LIN {X 0,Y 82.598,Z 477.464,A -85,B 0,C 180,E1 -27697.49,E2 -27697.49} C_VEL
LIN {X 0,Y 81.688,Z 489.871,A -85,B 0,C 180,E1 -27701.786,E2 -27701.786} C_VEL
LIN {X 0,Y 81.093,Z 501.439,A -85,B 0,C 180,E1 -27706.853,E2 -27706.853} C_VEL
LIN {X 0,Y 80.928,Z 512.952,A -85,B 0,C 180,E1 -27713.144,E2 -27713.144} C_VEL
LIN {X 0,Y 81.578,Z 523.458,A -85,B 0,C 180,E1 -27720.002,E2 -27720.002} C_VEL
LIN {X 0,Y 83.364,Z 532.882,A -85,B 0,C 180,E1 -27727.267,E2 -27727.267} C_VEL
LIN {X 0,Y 87.913,Z 543.523,A -85,B 0,C 180,E1 -27736.397,E2 -27736.397} C_VEL
LIN {X 0,Y 94.405,Z 551.821,A -85,B 0,C 180,E1 -27744.172,E2 -27744.172} C_VEL
LIN {X 0,Y 102.902,Z 558.75,A -85,B 0,C 180,E1 -27750.815,E2 -27750.815} C_VEL
LIN {X 0,Y 113.275,Z 564.386,A -85,B 0,C 180,E1 -27756.441,E2 -27756.441} C_VEL
LIN {X 0,Y 112.437,Z 564.55,A -85,B 0,C 180,E1 -27757.575,E2 -27757.575} C_VEL
LIN {X 0,Y 103.211,Z 562.875,A -85,B 0,C 180,E1 -27762.919,E2 -27762.919} C_VEL
LIN {X 0,Y 96.176,Z 560.643,A -85,B 0,C 180,E1 -27768.877,E2 -27768.877} C_VEL
LIN {X 0,Y 90.173,Z 557.258,A -85,B 0,C 180,E1 -27776.935,E2 -27776.935} C_VEL
LIN {X 0,Y 86.827,Z 552.894,A -85,B 0,C 180,E1 -27786.126,E2 -27786.126} C_VEL
LIN {X 0,Y 86.626,Z 546.753,A -85,B 0,C 180,E1 -27796.804,E2 -27796.804} C_VEL
LIN {X 0,Y 89.154,Z 540.243,A -85,B 0,C 180,E1 -27805.478,E2 -27805.478} C_VEL
LIN {X 0,Y 92.06,Z 533.359,A -85,B 0,C 180,E1 -27811.968,E2 -27811.968} C_VEL
LIN {X 0,Y 93.442,Z 531.34,A -85,B 0,C 180,E1 -27813.719,E2 -27813.719} C_VEL
LIN {X 0,Y 90.662,Z 537.837,A -85,B 0,C 180,E1 -27821.174,E2 -27821.174} C_VEL
LIN {X 0,Y 89.6,Z 544.588,A -85,B 0,C 180,E1 -27831.36,E2 -27831.36} C_VEL
LIN {X 0,Y 92.468,Z 550.453,A -85,B 0,C 180,E1 -27842.142,E2 -27842.142} C_VEL
LIN {X 0,Y 97.829,Z 554.403,A -85,B 0,C 180,E1 -27850.282,E2 -27850.282} C_VEL
LIN {X 0,Y 105.525,Z 557.586,A -85,B 0,C 180,E1 -27857.105,E2 -27857.105} C_VEL
LIN {X 0,Y 109.148,Z 558.477,A -85,B 0,C 180,E1 -27859.915,E2 -27859.915} C_VEL
LIN {X 0,Y 99.996,Z 550.972,A -85,B 0,C 180,E1 -27865.785,E2 -27865.785} C_VEL
LIN {X 0,Y 92.556,Z 542.014,A -85,B 0,C 180,E1 -27872.895,E2 -27872.895} C_VEL
LIN {X 0,Y 87.619,Z 532.647,A -85,B 0,C 180,E1 -27880.066,E2 -27880.066} C_VEL
LIN {X 0,Y 84.772,Z 523.292,A -85,B 0,C 180,E1 -27886.819,E2 -27886.819} C_VEL
LIN {X 0,Y 83.121,Z 511.282,A -85,B 0,C 180,E1 -27894.539,E2 -27894.539} C_VEL
LIN {X 0,Y 82.94,Z 507.215,A -85,B 0,C 180,E1 -27896.875,E2 -27896.875} C_VEL
LIN {X 0,Y 82.152,Z 502.38,A -85,B 0,C 180,E1 -27899.161,E2 -27899.161} C_VEL
LIN {X 0,Y 79.531,Z 493.78,A -85,B 0,C 180,E1 -27902.131,E2 -27902.131} C_VEL
LIN {X 0,Y 77.046,Z 484.849,A -85,B 0,C 180,E1 -27904.856,E2 -27904.856} C_VEL
LIN {X 0,Y 76.579,Z 479.375,A -85,B 0,C 180,E1 -27906.694,E2 -27906.694} C_VEL
LIN {X 0,Y 77.028,Z 465.248,A -85,B 0,C 180,E1 -27911.177,E2 -27911.177} C_VEL
LIN {X 0,Y 77.568,Z 451.467,A -85,B 0,C 180,E1 -27914.425,E2 -27914.425} C_VEL
LIN {X 0,Y 78.001,Z 427.384,A -85,B 0,C 180,E1 -27919.232,E2 -27919.232} C_VEL
LIN {X 0,Y 78.51,Z 395.761,A -85,B 0,C 180,E1 -27925.218,E2 -27925.218} C_VEL
LIN {X 0,Y 73.948,Z 377.278,A -85,B 0,C 180,E1 -27928.214,E2 -27928.214} C_VEL
LIN {X 0,Y 72.988,Z 372.385,A -85,B 0,C 180,E1 -27929.21,E2 -27929.21} C_VEL
LIN {X 0,Y 72.308,Z 372.47,A -85,B 0,C 180,E1 -27938.963,E2 -27938.963} C_VEL
LIN {X 0,Y 72.259,Z 372.475,A -85,B 0,C 180,E1 -27947.092,E2 -27947.092} C_VEL
LIN {X 0,Y 72.297,Z 372.472,A -85,B 0,C 180,E1 -27954.321,E2 -27954.321} C_VEL
LIN {X 0,Y 72.389,Z 372.467,A -85,B 0,C 180,E1 -27960.96,E2 -27960.96} C_VEL
LIN {X 0,Y 72.397,Z 372.466,A -85,B 0,C 180,E1 -27967.152,E2 -27967.152} C_VEL
LIN {X 0,Y 72.755,Z 372.419,A -85,B 0,C 180,E1 -27975.003,E2 -27975.003} C_VEL
LIN {X 0,Y 72.882,Z 372.404,A -85,B 0,C 180,E1 -27978.881,E2 -27978.881} C_VEL
LIN {X 0,Y 73.578,Z 372.311,A -85,B 0,C 180,E1 -27990.001,E2 -27990.001} C_VEL
LIN {X 0,Y 72.883,Z 372.405,A -85,B 0,C 180,E1 -28001.121,E2 -28001.121} C_VEL
LIN {X 0,Y 72.584,Z 372.435,A -85,B 0,C 180,E1 -28006.888,E2 -28006.888} C_VEL
LIN {X 0,Y 72.398,Z 372.465,A -85,B 0,C 180,E1 -28012.85,E2 -28012.85} C_VEL
LIN {X 0,Y 72.375,Z 372.469,A -85,B 0,C 180,E1 -28019.084,E2 -28019.084} C_VEL
LIN {X 0,Y 72.299,Z 372.474,A -85,B 0,C 180,E1 -28025.68,E2 -28025.68} C_VEL
LIN {X 0,Y 72.296,Z 372.471,A -85,B 0,C 180,E1 -28032.883,E2 -28032.883} C_VEL
LIN {X 0,Y 72.6,Z 372.44,A -85,B 0,C 180,E1 -28038.429,E2 -28038.429} C_VEL
LIN {X 0,Y 79.747,Z 400.874,A -85,B 0,C 180,E1 -28043.521,E2 -28043.521} C_VEL
LIN {X 0,Y 77.611,Z 449.683,A -85,B 0,C 180,E1 -28051.985,E2 -28051.985} C_VEL
LIN {X 0,Y 76.609,Z 464.552,A -85,B 0,C 180,E1 -28055.081,E2 -28055.081} C_VEL
LIN {X 0,Y 75.61,Z 478.192,A -85,B 0,C 180,E1 -28059.093,E2 -28059.093} C_VEL
LIN {X 0,Y 74.753,Z 491.561,A -85,B 0,C 180,E1 -28064.321,E2 -28064.321} C_VEL
LIN {X 0,Y 74.388,Z 502.747,A -85,B 0,C 180,E1 -28069.799,E2 -28069.799} C_VEL
LIN {X 0,Y 74.539,Z 514.065,A -85,B 0,C 180,E1 -28076.624,E2 -28076.624} C_VEL
LIN {X 0,Y 75.73,Z 524.288,A -85,B 0,C 180,E1 -28083.994,E2 -28083.994} C_VEL
LIN {X 0,Y 78.654,Z 535.064,A -85,B 0,C 180,E1 -28092.91,E2 -28092.91} C_VEL
LIN {X 0,Y 84.429,Z 545.209,A -85,B 0,C 180,E1 -28102.001,E2 -28102.001} C_VEL
LIN {X 0,Y 90.091,Z 551.599,A -85,B 0,C 180,E1 -28107.911,E2 -28107.911} C_VEL
LIN {X 0,Y 99.33,Z 558.739,A -85,B 0,C 180,E1 -28114.476,E2 -28114.476} C_VEL
LIN {X 0,Y 103.032,Z 560.997,A -85,B 0,C 180,E1 -28116.511,E2 -28116.511} C_VEL
LIN {X 0,Y 102.39,Z 561.181,A -85,B 0,C 180,E1 -28117.877,E2 -28117.877} C_VEL
LIN {X 0,Y 91.362,Z 557.787,A -85,B 0,C 180,E1 -28126.184,E2 -28126.184} C_VEL
LIN {X 0,Y 84.901,Z 554.088,A -85,B 0,C 180,E1 -28134.587,E2 -28134.587} C_VEL
LIN {X 0,Y 80.763,Z 548.053,A -85,B 0,C 180,E1 -28146.945,E2 -28146.945} C_VEL
LIN {X 0,Y 81.072,Z 541.907,A -85,B 0,C 180,E1 -28157.389,E2 -28157.389} C_VEL
LIN {X 0,Y 83.386,Z 536.089,A -85,B 0,C 180,E1 -28165.164,E2 -28165.164} C_VEL
LIN {X 0,Y 87.394,Z 527.549,A -85,B 0,C 180,E1 -28173.342,E2 -28173.342} C_VEL
LIN {X 0,Y 88.104,Z 526.717,A -85,B 0,C 180,E1 -28174.141,E2 -28174.141} C_VEL
LIN {X 0,Y 85.326,Z 533.18,A -85,B 0,C 180,E1 -28181.641,E2 -28181.641} C_VEL
LIN {X 0,Y 84.181,Z 539.373,A -85,B 0,C 180,E1 -28190.972,E2 -28190.972} C_VEL
LIN {X 0,Y 86.416,Z 545.437,A -85,B 0,C 180,E1 -28201.912,E2 -28201.912} C_VEL
LIN {X 0,Y 93.22,Z 550.858,A -85,B 0,C 180,E1 -28212.728,E2 -28212.728} C_VEL
LIN {X 0,Y 98.783,Z 553.406,A -85,B 0,C 180,E1 -28217.832,E2 -28217.832} C_VEL
LIN {X 0,Y 100.29,Z 553.807,A -85,B 0,C 180,E1 -28219.493,E2 -28219.493} C_VEL
LIN {X 0,Y 91.316,Z 545.13,A -85,B 0,C 180,E1 -28226.081,E2 -28226.081} C_VEL
LIN {X 0,Y 84.284,Z 534.916,A -85,B 0,C 180,E1 -28234.036,E2 -28234.036} C_VEL
LIN {X 0,Y 79.923,Z 524.257,A -85,B 0,C 180,E1 -28242.072,E2 -28242.072} C_VEL
LIN {X 0,Y 77.557,Z 513.408,A -85,B 0,C 180,E1 -28249.556,E2 -28249.556} C_VEL
LIN {X 0,Y 76.759,Z 503.923,A -85,B 0,C 180,E1 -28255.402,E2 -28255.402} C_VEL
LIN {X 0,Y 76.434,Z 492.423,A -85,B 0,C 180,E1 -28261.315,E2 -28261.315} C_VEL
LIN {X 0,Y 76.579,Z 479.375,A -85,B 0,C 180,E1 -28266.694,E2 -28266.694} C_VEL
LIN {X 0,Y 76.149,Z 474.078,A -85,B 0,C 180,E1 -28268.318,E2 -28268.318} C_VEL
LIN {X 0,Y 73.874,Z 464.959,A -85,B 0,C 180,E1 -28270.162,E2 -28270.162} C_VEL
LIN {X 0,Y 71.215,Z 453.2,A -85,B 0,C 180,E1 -28272.063,E2 -28272.063} C_VEL
LIN {X 0,Y 70.969,Z 449.25,A -85,B 0,C 180,E1 -28272.852,E2 -28272.852} C_VEL
LIN {X 0,Y 71.179,Z 426.045,A -85,B 0,C 180,E1 -28277.969,E2 -28277.969} C_VEL
LIN {X 0,Y 71.506,Z 396.594,A -85,B 0,C 180,E1 -28284.161,E2 -28284.161} C_VEL
LIN {X 0,Y 66.683,Z 376.694,A -85,B 0,C 180,E1 -28287.631,E2 -28287.631} C_VEL
LIN {X 0,Y 66.023,Z 373.254,A -85,B 0,C 180,E1 -28288.427,E2 -28288.427} C_VEL
LIN {X 0,Y 65.197,Z 373.361,A -85,B 0,C 180,E1 -28301.013,E2 -28301.013} C_VEL
LIN {X 0,Y 65.209,Z 373.36,A -85,B 0,C 180,E1 -28309.711,E2 -28309.711} C_VEL
LIN {X 0,Y 65.252,Z 373.357,A -85,B 0,C 180,E1 -28319.496,E2 -28319.496} C_VEL
LIN {X 0,Y 65.245,Z 373.349,A -85,B 0,C 180,E1 -28324.478,E2 -28324.478} C_VEL
LIN {X 0,Y 65.649,Z 373.302,A -85,B 0,C 180,E1 -28334.459,E2 -28334.459} C_VEL
LIN {X 0,Y 65.781,Z 373.291,A -85,B 0,C 180,E1 -28337.663,E2 -28337.663} C_VEL
LIN {X 0,Y 66.503,Z 373.192,A -85,B 0,C 180,E1 -28350.001,E2 -28350.001} C_VEL
LIN {X 0,Y 65.781,Z 373.291,A -85,B 0,C 180,E1 -28362.339,E2 -28362.339} C_VEL
LIN {X 0,Y 65.388,Z 373.335,A -85,B 0,C 180,E1 -28368.812,E2 -28368.812} C_VEL
LIN {X 0,Y 65.247,Z 373.348,A -85,B 0,C 180,E1 -28375.523,E2 -28375.523} C_VEL
LIN {X 0,Y 65.197,Z 373.357,A -85,B 0,C 180,E1 -28382.616,E2 -28382.616} C_VEL
LIN {X 0,Y 65.214,Z 373.356,A -85,B 0,C 180,E1 -28391.033,E2 -28391.033} C_VEL
LIN {X 0,Y 65.558,Z 373.317,A -85,B 0,C 180,E1 -28398.208,E2 -28398.208} C_VEL
LIN {X 0,Y 71.869,Z 398.471,A -85,B 0,C 180,E1 -28403.177,E2 -28403.177} C_VEL
LIN {X 0,Y 72.589,Z 400.996,A -85,B 0,C 180,E1 -28403.632,E2 -28403.632} C_VEL
LIN {X 0,Y 70.68,Z 448.813,A -85,B 0,C 180,E1 -28412.864,E2 -28412.864} C_VEL
LIN {X 0,Y 69.712,Z 464.246,A -85,B 0,C 180,E1 -28416.409,E2 -28416.409} C_VEL
LIN {X 0,Y 68.738,Z 478.221,A -85,B 0,C 180,E1 -28420.889,E2 -28420.889} C_VEL
LIN {X 0,Y 68.061,Z 491.519,A -85,B 0,C 180,E1 -28426.568,E2 -28426.568} C_VEL
LIN {X 0,Y 67.911,Z 502.664,A -85,B 0,C 180,E1 -28432.57,E2 -28432.57} C_VEL
LIN {X 0,Y 68.396,Z 513.871,A -85,B 0,C 180,E1 -28440.003,E2 -28440.003} C_VEL
LIN {X 0,Y 70.213,Z 525.012,A -85,B 0,C 180,E1 -28448.638,E2 -28448.638} C_VEL
LIN {X 0,Y 74.374,Z 536.126,A -85,B 0,C 180,E1 -28458.405,E2 -28458.405} C_VEL
LIN {X 0,Y 79.979,Z 544.629,A -85,B 0,C 180,E1 -28466.066,E2 -28466.066} C_VEL
LIN {X 0,Y 88.569,Z 553.193,A -85,B 0,C 180,E1 -28473.744,E2 -28473.744} C_VEL
LIN {X 0,Y 93.544,Z 556.898,A -85,B 0,C 180,E1 -28476.947,E2 -28476.947} C_VEL
LIN {X 0,Y 91.184,Z 556.389,A -85,B 0,C 180,E1 -28479.577,E2 -28479.577} C_VEL
LIN {X 0,Y 83.059,Z 552.829,A -85,B 0,C 180,E1 -28487.396,E2 -28487.396} C_VEL
LIN {X 0,Y 77.437,Z 548.364,A -85,B 0,C 180,E1 -28497.005,E2 -28497.005} C_VEL
LIN {X 0,Y 74.907,Z 541.807,A -85,B 0,C 180,E1 -28509.764,E2 -28509.764} C_VEL
LIN {X 0,Y 76.478,Z 534.839,A -85,B 0,C 180,E1 -28520.878,E2 -28520.878} C_VEL
LIN {X 0,Y 78.232,Z 530.448,A -85,B 0,C 180,E1 -28526.269,E2 -28526.269} C_VEL
LIN {X 0,Y 81.23,Z 524.037,A -85,B 0,C 180,E1 -28532.41,E2 -28532.41} C_VEL
LIN {X 0,Y 82.901,Z 521.941,A -85,B 0,C 180,E1 -28534.549,E2 -28534.549} C_VEL
LIN {X 0,Y 80.02,Z 528.732,A -85,B 0,C 180,E1 -28542.686,E2 -28542.686} C_VEL
LIN {X 0,Y 79.069,Z 535.662,A -85,B 0,C 180,E1 -28553.601,E2 -28553.601} C_VEL
LIN {X 0,Y 81.547,Z 541.351,A -85,B 0,C 180,E1 -28564.068,E2 -28564.068} C_VEL
LIN {X 0,Y 87.28,Z 546.183,A -85,B 0,C 180,E1 -28573.553,E2 -28573.553} C_VEL
LIN {X 0,Y 88.875,Z 547.115,A -85,B 0,C 180,E1 -28575.372,E2 -28575.372} C_VEL
LIN {X 0,Y 91.443,Z 548.021,A -85,B 0,C 180,E1 -28579.208,E2 -28579.208} C_VEL
LIN {X 0,Y 82.894,Z 538.278,A -85,B 0,C 180,E1 -28586.556,E2 -28586.556} C_VEL
LIN {X 0,Y 76.975,Z 528.208,A -85,B 0,C 180,E1 -28594.295,E2 -28594.295} C_VEL
LIN {X 0,Y 73.396,Z 518.149,A -85,B 0,C 180,E1 -28601.866,E2 -28601.866} C_VEL
LIN {X 0,Y 71.141,Z 504.498,A -85,B 0,C 180,E1 -28611.189,E2 -28611.189} C_VEL
LIN {X 0,Y 70.427,Z 492.689,A -85,B 0,C 180,E1 -28617.853,E2 -28617.853} C_VEL
LIN {X 0,Y 70.233,Z 480.023,A -85,B 0,C 180,E1 -28623.583,E2 -28623.583} C_VEL
LIN {X 0,Y 70.469,Z 467.033,A -85,B 0,C 180,E1 -28628.24,E2 -28628.24} C_VEL
LIN {X 0,Y 70.944,Z 452.368,A -85,B 0,C 180,E1 -28632.15,E2 -28632.15} C_VEL
LIN {X 0,Y 70.969,Z 449.25,A -85,B 0,C 180,E1 -28632.852,E2 -28632.852} C_VEL
LIN {X 0,Y 70.415,Z 443.52,A -85,B 0,C 180,E1 -28633.947,E2 -28633.947} C_VEL
LIN {X 0,Y 64.964,Z 424.632,A -85,B 0,C 180,E1 -28636.547,E2 -28636.547} C_VEL
LIN {X 0,Y 64.297,Z 418.882,A -85,B 0,C 180,E1 -28637.703,E2 -28637.703} C_VEL
LIN {X 0,Y 64.462,Z 396.873,A -85,B 0,C 180,E1 -28642.867,E2 -28642.867} C_VEL
LIN {X 0,Y 59.791,Z 377.73,A -85,B 0,C 180,E1 -28646.465,E2 -28646.465} C_VEL
LIN {X 0,Y 59.094,Z 374.122,A -85,B 0,C 180,E1 -28647.312,E2 -28647.312} C_VEL
LIN {X 0,Y 58.176,Z 374.231,A -85,B 0,C 180,E1 -28657.154,E2 -28657.154} C_VEL
LIN {X 0,Y 58.02,Z 374.249,A -85,B 0,C 180,E1 -28666.612,E2 -28666.612} C_VEL
LIN {X 0,Y 58.035,Z 374.254,A -85,B 0,C 180,E1 -28672.736,E2 -28672.736} C_VEL
LIN {X 0,Y 58.151,Z 374.24,A -85,B 0,C 180,E1 -28681.092,E2 -28681.092} C_VEL
LIN {X 0,Y 58.535,Z 374.186,A -85,B 0,C 180,E1 -28693.835,E2 -28693.835} C_VEL
LIN {X 0,Y 58.822,Z 374.152,A -85,B 0,C 180,E1 -28703.139,E2 -28703.139} C_VEL
LIN {X 0,Y 59.395,Z 374.077,A -85,B 0,C 180,E1 -28710.001,E2 -28710.001} C_VEL
LIN {X 0,Y 58.822,Z 374.151,A -85,B 0,C 180,E1 -28716.863,E2 -28716.863} C_VEL
LIN {X 0,Y 58.535,Z 374.185,A -85,B 0,C 180,E1 -28726.167,E2 -28726.167} C_VEL
LIN {X 0,Y 58.153,Z 374.241,A -85,B 0,C 180,E1 -28738.91,E2 -28738.91} C_VEL
LIN {X 0,Y 58.046,Z 374.254,A -85,B 0,C 180,E1 -28747.258,E2 -28747.258} C_VEL
LIN {X 0,Y 58.484,Z 374.22,A -85,B 0,C 180,E1 -28758.198,E2 -28758.198} C_VEL
LIN {X 0,Y 64.852,Z 399.555,A -85,B 0,C 180,E1 -28763.636,E2 -28763.636} C_VEL
LIN {X 0,Y 65.427,Z 402.184,A -85,B 0,C 180,E1 -28764.147,E2 -28764.147} C_VEL
LIN {X 0,Y 63.761,Z 448.002,A -85,B 0,C 180,E1 -28774.051,E2 -28774.051} C_VEL
LIN {X 0,Y 62.812,Z 464.656,A -85,B 0,C 180,E1 -28778.269,E2 -28778.269} C_VEL
LIN {X 0,Y 62.044,Z 477.202,A -85,B 0,C 180,E1 -28782.705,E2 -28782.705} C_VEL
LIN {X 0,Y 61.546,Z 489.628,A -85,B 0,C 180,E1 -28788.476,E2 -28788.476} C_VEL
LIN {X 0,Y 61.677,Z 502.331,A -85,B 0,C 180,E1 -28795.919,E2 -28795.919} C_VEL
LIN {X 0,Y 62.551,Z 513.655,A -85,B 0,C 180,E1 -28804.03,E2 -28804.03} C_VEL
LIN {X 0,Y 64.893,Z 524.229,A -85,B 0,C 180,E1 -28812.905,E2 -28812.905} C_VEL
LIN {X 0,Y 69.442,Z 534.827,A -85,B 0,C 180,E1 -28822.402,E2 -28822.402} C_VEL
LIN {X 0,Y 76.021,Z 543.908,A -85,B 0,C 180,E1 -28830.564,E2 -28830.564} C_VEL
LIN {X 0,Y 84.922,Z 552.311,A -85,B 0,C 180,E1 -28837.791,E2 -28837.791} C_VEL
LIN {X 0,Y 80.555,Z 550.429,A -85,B 0,C 180,E1 -28842.132,E2 -28842.132} C_VEL
LIN {X 0,Y 73.865,Z 546.009,A -85,B 0,C 180,E1 -28851.417,E2 -28851.417} C_VEL
LIN {X 0,Y 69.976,Z 540.311,A -85,B 0,C 180,E1 -28863.133,E2 -28863.133} C_VEL
LIN {X 0,Y 69.955,Z 533.424,A -85,B 0,C 180,E1 -28875.605,E2 -28875.605} C_VEL
LIN {X 0,Y 72.264,Z 527.154,A -85,B 0,C 180,E1 -28884.418,E2 -28884.418} C_VEL
LIN {X 0,Y 75.177,Z 520.459,A -85,B 0,C 180,E1 -28891.34,E2 -28891.34} C_VEL
LIN {X 0,Y 77.971,Z 516.858,A -85,B 0,C 180,E1 -28894.88,E2 -28894.88} C_VEL
LIN {X 0,Y 74.982,Z 523.867,A -85,B 0,C 180,E1 -28903.554,E2 -28903.554} C_VEL
LIN {X 0,Y 74.128,Z 531.106,A -85,B 0,C 180,E1 -28915.281,E2 -28915.281} C_VEL
LIN {X 0,Y 76.944,Z 537.055,A -85,B 0,C 180,E1 -28926.419,E2 -28926.419} C_VEL
LIN {X 0,Y 81.175,Z 540.859,A -85,B 0,C 180,E1 -28933.838,E2 -28933.838} C_VEL
LIN {X 0,Y 84.094,Z 542.571,A -85,B 0,C 180,E1 -28938.039,E2 -28938.039} C_VEL
LIN {X 0,Y 75.642,Z 531.766,A -85,B 0,C 180,E1 -28946.116,E2 -28946.116} C_VEL
LIN {X 0,Y 69.917,Z 520.434,A -85,B 0,C 180,E1 -28954.864,E2 -28954.864} C_VEL
LIN {X 0,Y 66.476,Z 508.18,A -85,B 0,C 180,E1 -28963.885,E2 -28963.885} C_VEL
LIN {X 0,Y 65.246,Z 499.423,A -85,B 0,C 180,E1 -28969.752,E2 -28969.752} C_VEL
LIN {X 0,Y 64.476,Z 488.384,A -85,B 0,C 180,E1 -28976.091,E2 -28976.091} C_VEL
LIN {X 0,Y 64.181,Z 474.703,A -85,B 0,C 180,E1 -28982.35,E2 -28982.35} C_VEL
LIN {X 0,Y 64.338,Z 460.673,A -85,B 0,C 180,E1 -28987.254,E2 -28987.254} C_VEL
LIN {X 0,Y 64.533,Z 442.476,A -85,B 0,C 180,E1 -28992.039,E2 -28992.039} C_VEL
LIN {X 0,Y 64.304,Z 419.795,A -85,B 0,C 180,E1 -28997.488,E2 -28997.488} C_VEL
LIN {X 0,Y 64.297,Z 418.882,A -85,B 0,C 180,E1 -28997.703,E2 -28997.703} C_VEL
LIN {X 0,Y 63.654,Z 413.138,A -85,B 0,C 180,E1 -28998.884,E2 -28998.884} C_VEL
LIN {X 0,Y 62.061,Z 407.479,A -85,B 0,C 180,E1 -28999.801,E2 -28999.801} C_VEL
LIN {X 0,Y 57.694,Z 396.336,A -85,B 0,C 180,E1 -29001.397,E2 -29001.397} C_VEL
LIN {X 0,Y 55.264,Z 388.755,A -85,B 0,C 180,E1 -29002.738,E2 -29002.738} C_VEL
LIN {X 0,Y 52.196,Z 374.983,A -85,B 0,C 180,E1 -29005.938,E2 -29005.938} C_VEL
LIN {X 0,Y 51.249,Z 375.101,A -85,B 0,C 180,E1 -29014.635,E2 -29014.635} C_VEL
LIN {X 0,Y 50.987,Z 375.125,A -85,B 0,C 180,E1 -29026.435,E2 -29026.435} C_VEL
LIN {X 0,Y 51.05,Z 375.117,A -85,B 0,C 180,E1 -29036.588,E2 -29036.588} C_VEL
LIN {X 0,Y 51.025,Z 375.121,A -85,B 0,C 180,E1 -29045.595,E2 -29045.595} C_VEL
LIN {X 0,Y 51.479,Z 375.065,A -85,B 0,C 180,E1 -29054.156,E2 -29054.156} C_VEL
LIN {X 0,Y 51.698,Z 375.036,A -85,B 0,C 180,E1 -29062.188,E2 -29062.188} C_VEL
LIN {X 0,Y 52.28,Z 374.963,A -85,B 0,C 180,E1 -29070.001,E2 -29070.001} C_VEL
LIN {X 0,Y 51.698,Z 375.036,A -85,B 0,C 180,E1 -29077.815,E2 -29077.815} C_VEL
LIN {X 0,Y 51.401,Z 375.072,A -85,B 0,C 180,E1 -29086.858,E2 -29086.858} C_VEL
LIN {X 0,Y 51.027,Z 375.12,A -85,B 0,C 180,E1 -29094.407,E2 -29094.407} C_VEL
LIN {X 0,Y 51.034,Z 375.118,A -85,B 0,C 180,E1 -29104.288,E2 -29104.288} C_VEL
LIN {X 0,Y 51.434,Z 375.077,A -85,B 0,C 180,E1 -29118.102,E2 -29118.102} C_VEL
LIN {X 0,Y 57.715,Z 400.202,A -85,B 0,C 180,E1 -29124.151,E2 -29124.151} C_VEL
LIN {X 0,Y 58.338,Z 402.3,A -85,B 0,C 180,E1 -29124.596,E2 -29124.596} C_VEL
LIN {X 0,Y 56.895,Z 447.294,A -85,B 0,C 180,E1 -29135.608,E2 -29135.608} C_VEL
LIN {X 0,Y 56.057,Z 465.197,A -85,B 0,C 180,E1 -29140.789,E2 -29140.789} C_VEL
LIN {X 0,Y 55.403,Z 478.522,A -85,B 0,C 180,E1 -29146.244,E2 -29146.244} C_VEL
LIN {X 0,Y 55.223,Z 490.748,A -85,B 0,C 180,E1 -29152.692,E2 -29152.692} C_VEL
LIN {X 0,Y 55.684,Z 501.908,A -85,B 0,C 180,E1 -29160.003,E2 -29160.003} C_VEL
LIN {X 0,Y 57.339,Z 514.092,A -85,B 0,C 180,E1 -29169.706,E2 -29169.706} C_VEL
LIN {X 0,Y 60.562,Z 524.847,A -85,B 0,C 180,E1 -29179.243,E2 -29179.243} C_VEL
LIN {X 0,Y 67.124,Z 536.432,A -85,B 0,C 180,E1 -29189.827,E2 -29189.827} C_VEL
LIN {X 0,Y 74.83,Z 545.302,A -85,B 0,C 180,E1 -29197.442,E2 -29197.442} C_VEL
LIN {X 0,Y 76.156,Z 546.519,A -85,B 0,C 180,E1 -29198.455,E2 -29198.455} C_VEL
LIN {X 0,Y 73.698,Z 545.319,A -85,B 0,C 180,E1 -29201.88,E2 -29201.88} C_VEL
LIN {X 0,Y 67.743,Z 540.69,A -85,B 0,C 180,E1 -29211.502,E2 -29211.502} C_VEL
LIN {X 0,Y 64.454,Z 534.562,A -85,B 0,C 180,E1 -29224.14,E2 -29224.14} C_VEL
LIN {X 0,Y 65.197,Z 527.04,A -85,B 0,C 180,E1 -29237.549,E2 -29237.549} C_VEL
LIN {X 0,Y 66.937,Z 522.349,A -85,B 0,C 180,E1 -29243.972,E2 -29243.972} C_VEL
LIN {X 0,Y 70.319,Z 515.053,A -85,B 0,C 180,E1 -29251.829,E2 -29251.829} C_VEL
LIN {X 0,Y 73.169,Z 511.664,A -85,B 0,C 180,E1 -29255.338,E2 -29255.338} C_VEL
LIN {X 0,Y 69.83,Z 519.827,A -85,B 0,C 180,E1 -29266.068,E2 -29266.068} C_VEL
LIN {X 0,Y 69.423,Z 526.324,A -85,B 0,C 180,E1 -29277.1,E2 -29277.1} C_VEL
LIN {X 0,Y 72.834,Z 532.816,A -85,B 0,C 180,E1 -29289.467,E2 -29289.467} C_VEL
LIN {X 0,Y 75.484,Z 535.301,A -85,B 0,C 180,E1 -29294.289,E2 -29294.289} C_VEL
LIN {X 0,Y 76.522,Z 535.775,A -85,B 0,C 180,E1 -29297.23,E2 -29297.23} C_VEL
LIN {X 0,Y 69.535,Z 526.007,A -85,B 0,C 180,E1 -29304.464,E2 -29304.464} C_VEL
LIN {X 0,Y 64.32,Z 515.117,A -85,B 0,C 180,E1 -29312.87,E2 -29312.87} C_VEL
LIN {X 0,Y 60.746,Z 501.837,A -85,B 0,C 180,E1 -29322.751,E2 -29322.751} C_VEL
LIN {X 0,Y 59.151,Z 489.4,A -85,B 0,C 180,E1 -29330.765,E2 -29330.765} C_VEL
LIN {X 0,Y 58.356,Z 476.494,A -85,B 0,C 180,E1 -29337.408,E2 -29337.408} C_VEL
LIN {X 0,Y 58.157,Z 464.381,A -85,B 0,C 180,E1 -29342.377,E2 -29342.377} C_VEL
LIN {X 0,Y 58.234,Z 450.002,A -85,B 0,C 180,E1 -29346.928,E2 -29346.928} C_VEL
LIN {X 0,Y 57.841,Z 425.985,A -85,B 0,C 180,E1 -29353.583,E2 -29353.583} C_VEL
LIN {X 0,Y 57.625,Z 397.528,A -85,B 0,C 180,E1 -29361.074,E2 -29361.074} C_VEL
LIN {X 0,Y 55.264,Z 388.755,A -85,B 0,C 180,E1 -29362.738,E2 -29362.738} C_VEL
LIN {X 0,Y 54.035,Z 385.432,A -85,B 0,C 180,E1 -29363.984,E2 -29363.984} C_VEL
LIN {X 0,Y 52.302,Z 382.688,A -85,B 0,C 180,E1 -29366.054,E2 -29366.054} C_VEL
LIN {X 0,Y 49.36,Z 379.59,A -85,B 0,C 180,E1 -29370.453,E2 -29370.453} C_VEL
LIN {X 0,Y 46.561,Z 377.565,A -85,B 0,C 180,E1 -29376.393,E2 -29376.393} C_VEL
LIN {X 0,Y 44.525,Z 376.403,A -85,B 0,C 180,E1 -29383.596,E2 -29383.596} C_VEL
LIN {X 0,Y 43.805,Z 376.022,A -85,B 0,C 180,E1 -29391.549,E2 -29391.549} C_VEL
LIN {X 0,Y 43.843,Z 376.021,A -85,B 0,C 180,E1 -29401.258,E2 -29401.258} C_VEL
LIN {X 0,Y 44.255,Z 375.963,A -85,B 0,C 180,E1 -29412.32,E2 -29412.32} C_VEL
LIN {X 0,Y 44.55,Z 375.926,A -85,B 0,C 180,E1 -29420.925,E2 -29420.925} C_VEL
LIN {X 0,Y 45.155,Z 375.85,A -85,B 0,C 180,E1 -29430.002,E2 -29430.002} C_VEL
LIN {X 0,Y 44.55,Z 375.926,A -85,B 0,C 180,E1 -29439.078,E2 -29439.078} C_VEL
LIN {X 0,Y 44.192,Z 375.972,A -85,B 0,C 180,E1 -29448.548,E2 -29448.548} C_VEL
LIN {X 0,Y 43.838,Z 376.023,A -85,B 0,C 180,E1 -29458.75,E2 -29458.75} C_VEL
LIN {X 0,Y 43.912,Z 376.012,A -85,B 0,C 180,E1 -29469.808,E2 -29469.808} C_VEL
LIN {X 0,Y 44.379,Z 376.021,A -85,B 0,C 180,E1 -29478.357,E2 -29478.357} C_VEL
LIN {X 0,Y 50.662,Z 401.016,A -85,B 0,C 180,E1 -29485.021,E2 -29485.021} C_VEL
LIN {X 0,Y 51.189,Z 403.547,A -85,B 0,C 180,E1 -29485.625,E2 -29485.625} C_VEL
LIN {X 0,Y 50.13,Z 446.886,A -85,B 0,C 180,E1 -29497.87,E2 -29497.87} C_VEL
LIN {X 0,Y 49.457,Z 464.871,A -85,B 0,C 180,E1 -29503.758,E2 -29503.758} C_VEL
LIN {X 0,Y 49.006,Z 479.785,A -85,B 0,C 180,E1 -29510.719,E2 -29510.719} C_VEL
LIN {X 0,Y 49.351,Z 492.748,A -85,B 0,C 180,E1 -29518.779,E2 -29518.779} C_VEL
LIN {X 0,Y 50.418,Z 503.481,A -85,B 0,C 180,E1 -29526.911,E2 -29526.911} C_VEL
LIN {X 0,Y 53.135,Z 515.549,A -85,B 0,C 180,E1 -29537.355,E2 -29537.355} C_VEL
LIN {X 0,Y 58.565,Z 527.676,A -85,B 0,C 180,E1 -29548.69,E2 -29548.69} C_VEL
LIN {X 0,Y 64.9,Z 536.629,A -85,B 0,C 180,E1 -29556.559,E2 -29556.559} C_VEL
LIN {X 0,Y 68.101,Z 540.183,A -85,B 0,C 180,E1 -29559.494,E2 -29559.494} C_VEL
LIN {X 0,Y 67.525,Z 539.972,A -85,B 0,C 180,E1 -29561.171,E2 -29561.171} C_VEL
LIN {X 0,Y 61.344,Z 534.134,A -85,B 0,C 180,E1 -29573.323,E2 -29573.323} C_VEL
LIN {X 0,Y 59.192,Z 528.037,A -85,B 0,C 180,E1 -29585.943,E2 -29585.943} C_VEL
LIN {X 0,Y 60.679,Z 520.455,A -85,B 0,C 180,E1 -29599.31,E2 -29599.31} C_VEL
LIN {X 0,Y 64.286,Z 511.561,A -85,B 0,C 180,E1 -29609.999,E2 -29609.999} C_VEL
LIN {X 0,Y 68.535,Z 506.314,A -85,B 0,C 180,E1 -29615.7,E2 -29615.7} C_VEL
LIN {X 0,Y 64.981,Z 515.662,A -85,B 0,C 180,E1 -29628.932,E2 -29628.932} C_VEL
LIN {X 0,Y 65.523,Z 523.102,A -85,B 0,C 180,E1 -29642.431,E2 -29642.431} C_VEL
LIN {X 0,Y 70.026,Z 529.296,A -85,B 0,C 180,E1 -29654.63,E2 -29654.63} C_VEL
LIN {X 0,Y 70.172,Z 529.325,A -85,B 0,C 180,E1 -29655.483,E2 -29655.483} C_VEL
LIN {X 0,Y 62.749,Z 517.834,A -85,B 0,C 180,E1 -29663.98,E2 -29663.98} C_VEL
LIN {X 0,Y 58.164,Z 507.099,A -85,B 0,C 180,E1 -29672.2,E2 -29672.2} C_VEL
LIN {X 0,Y 55.382,Z 495.976,A -85,B 0,C 180,E1 -29680.539,E2 -29680.539} C_VEL
LIN {X 0,Y 53.776,Z 484.774,A -85,B 0,C 180,E1 -29687.735,E2 -29687.735} C_VEL
LIN {X 0,Y 52.736,Z 471.356,A -85,B 0,C 180,E1 -29694.74,E2 -29694.74} C_VEL
LIN {X 0,Y 52.388,Z 456.383,A -85,B 0,C 180,E1 -29700.717,E2 -29700.717} C_VEL
LIN {X 0,Y 51.62,Z 430.662,A -85,B 0,C 180,E1 -29708.955,E2 -29708.955} C_VEL
LIN {X 0,Y 50.695,Z 397.579,A -85,B 0,C 180,E1 -29718.786,E2 -29718.786} C_VEL
LIN {X 0,Y 45.661,Z 377.499,A -85,B 0,C 180,E1 -29723.222,E2 -29723.222} C_VEL
LIN {X 0,Y 45.372,Z 375.83,A -85,B 0,C 180,E1 -29723.844,E2 -29723.844} C_VEL
LIN {X 0,Y 43.916,Z 376.006,A -85,B 0,C 180,E1 -29739.796,E2 -29739.796} C_VEL
LIN {X 0,Y 43.805,Z 376.022,A -85,B 0,C 180,E1 -29751.549,E2 -29751.549} C_VEL
LIN {X 0,Y 43.203,Z 376.1,A -85,B 0,C 180,E1 -29756.594,E2 -29756.594} C_VEL
LIN {X 0,Y 41.762,Z 376.291,A -85,B 0,C 180,E1 -29761.562,E2 -29761.562} C_VEL
LIN {X 0,Y 37.405,Z 376.821,A -85,B 0,C 180,E1 -29778.462,E2 -29778.462} C_VEL
LIN {X 0,Y 37.357,Z 376.815,A -85,B 0,C 180,E1 -29780.589,E2 -29780.589} C_VEL
LIN {X 0,Y 38.014,Z 376.74,A -85,B 0,C 180,E1 -29790.002,E2 -29790.002} C_VEL
LIN {X 0,Y 37.347,Z 376.827,A -85,B 0,C 180,E1 -29800.848,E2 -29800.848} C_VEL
LIN {X 0,Y 37.078,Z 376.858,A -85,B 0,C 180,E1 -29808.621,E2 -29808.621} C_VEL
LIN {X 0,Y 36.762,Z 376.896,A -85,B 0,C 180,E1 -29824.999,E2 -29824.999} C_VEL
LIN {X 0,Y 37.317,Z 376.831,A -85,B 0,C 180,E1 -29838.541,E2 -29838.541} C_VEL
LIN {X 0,Y 43.94,Z 402.921,A -85,B 0,C 180,E1 -29846.579,E2 -29846.579} C_VEL
LIN {X 0,Y 43.876,Z 408.91,A -85,B 0,C 180,E1 -29848.454,E2 -29848.454} C_VEL
LIN {X 0,Y 43.5,Z 445.648,A -85,B 0,C 180,E1 -29860.54,E2 -29860.54} C_VEL
LIN {X 0,Y 43.088,Z 464.346,A -85,B 0,C 180,E1 -29867.718,E2 -29867.718} C_VEL
LIN {X 0,Y 43.004,Z 476.758,A -85,B 0,C 180,E1 -29874.142,E2 -29874.142} C_VEL
LIN {X 0,Y 43.722,Z 490.644,A -85,B 0,C 180,E1 -29883.46,E2 -29883.46} C_VEL
LIN {X 0,Y 45.158,Z 501.035,A -85,B 0,C 180,E1 -29891.828,E2 -29891.828} C_VEL
LIN {X 0,Y 48.405,Z 512.669,A -85,B 0,C 180,E1 -29902.408,E2 -29902.408} C_VEL
LIN {X 0,Y 54.171,Z 524.533,A -85,B 0,C 180,E1 -29913.466,E2 -29913.466} C_VEL
LIN {X 0,Y 59.854,Z 532.34,A -85,B 0,C 180,E1 -29920.23,E2 -29920.23} C_VEL
LIN {X 0,Y 60.536,Z 533.334,A -85,B 0,C 180,E1 -29922.295,E2 -29922.295} C_VEL
LIN {X 0,Y 55.311,Z 526.754,A -85,B 0,C 180,E1 -29936.321,E2 -29936.321} C_VEL
LIN {X 0,Y 54.467,Z 520.357,A -85,B 0,C 180,E1 -29949.611,E2 -29949.611} C_VEL
LIN {X 0,Y 56.09,Z 514.142,A -85,B 0,C 180,E1 -29960.106,E2 -29960.106} C_VEL
LIN {X 0,Y 58.647,Z 507.606,A -85,B 0,C 180,E1 -29968.243,E2 -29968.243} C_VEL
LIN {X 0,Y 62.342,Z 502.402,A -85,B 0,C 180,E1 -29974.153,E2 -29974.153} C_VEL
LIN {X 0,Y 64.328,Z 500.635,A -85,B 0,C 180,E1 -29976.271,E2 -29976.271} C_VEL
LIN {X 0,Y 61.582,Z 506.245,A -85,B 0,C 180,E1 -29984.078,E2 -29984.078} C_VEL
LIN {X 0,Y 60.312,Z 513.099,A -85,B 0,C 180,E1 -29995.471,E2 -29995.471} C_VEL
LIN {X 0,Y 62.684,Z 520.331,A -85,B 0,C 180,E1 -30009.608,E2 -30009.608} C_VEL
LIN {X 0,Y 63.455,Z 521.369,A -85,B 0,C 180,E1 -30011.646,E2 -30011.646} C_VEL
LIN {X 0,Y 63.601,Z 521.429,A -85,B 0,C 180,E1 -30014.035,E2 -30014.035} C_VEL
LIN {X 0,Y 56.22,Z 508.564,A -85,B 0,C 180,E1 -30023.569,E2 -30023.569} C_VEL
LIN {X 0,Y 51.621,Z 495.268,A -85,B 0,C 180,E1 -30033.734,E2 -30033.734} C_VEL
LIN {X 0,Y 49.11,Z 482.633,A -85,B 0,C 180,E1 -30042.292,E2 -30042.292} C_VEL
LIN {X 0,Y 47.566,Z 468.146,A -85,B 0,C 180,E1 -30050.159,E2 -30050.159} C_VEL
LIN {X 0,Y 46.693,Z 450.947,A -85,B 0,C 180,E1 -30057.3,E2 -30057.3} C_VEL
LIN {X 0,Y 45.307,Z 426.616,A -85,B 0,C 180,E1 -30065.838,E2 -30065.838} C_VEL
LIN {X 0,Y 44.048,Z 397.94,A -85,B 0,C 180,E1 -30075.604,E2 -30075.604} C_VEL
LIN {X 0,Y 38.835,Z 377.449,A -85,B 0,C 180,E1 -30080.462,E2 -30080.462} C_VEL
LIN {X 0,Y 38.656,Z 376.66,A -85,B 0,C 180,E1 -30080.939,E2 -30080.939} C_VEL
LIN {X 0,Y 36.807,Z 376.892,A -85,B 0,C 180,E1 -30100.206,E2 -30100.206} C_VEL
LIN {X 0,Y 36.701,Z 376.904,A -85,B 0,C 180,E1 -30111.338,E2 -30111.338} C_VEL
LIN {X 0,Y 36.721,Z 376.901,A -85,B 0,C 180,E1 -30114.961,E2 -30114.961} C_VEL
LIN {X 0,Y 37.077,Z 376.857,A -85,B 0,C 180,E1 -30131.38,E2 -30131.38} C_VEL
LIN {X 0,Y 37.357,Z 376.815,A -85,B 0,C 180,E1 -30140.589,E2 -30140.589} C_VEL
LIN {X 0,Y 36.887,Z 376.891,A -85,B 0,C 180,E1 -30145.474,E2 -30145.474} C_VEL
LIN {X 0,Y 35.075,Z 377.114,A -85,B 0,C 180,E1 -30152.169,E2 -30152.169} C_VEL
LIN {X 0,Y 29.759,Z 377.649,A -85,B 0,C 180,E1 -30172.542,E2 -30172.542} C_VEL
LIN {X 0,Y 29.598,Z 377.657,A -85,B 0,C 180,E1 -30175.264,E2 -30175.264} C_VEL
LIN {X 0,Y 30.011,Z 377.625,A -85,B 0,C 180,E1 -30195.378,E2 -30195.378} C_VEL
LIN {X 0,Y 30.253,Z 377.601,A -85,B 0,C 180,E1 -30199.263,E2 -30199.263} C_VEL
LIN {X 0,Y 36.87,Z 403.378,A -85,B 0,C 180,E1 -30208.414,E2 -30208.414} C_VEL
LIN {X 0,Y 36.925,Z 408.58,A -85,B 0,C 180,E1 -30210.352,E2 -30210.352} C_VEL
LIN {X 0,Y 37.085,Z 445.333,A -85,B 0,C 180,E1 -30224.866,E2 -30224.866} C_VEL
LIN {X 0,Y 37.067,Z 463.179,A -85,B 0,C 180,E1 -30232.858,E2 -30232.858} C_VEL
LIN {X 0,Y 37.407,Z 476.799,A -85,B 0,C 180,E1 -30240.873,E2 -30240.873} C_VEL
LIN {X 0,Y 38.514,Z 488.183,A -85,B 0,C 180,E1 -30249.299,E2 -30249.299} C_VEL
LIN {X 0,Y 40.724,Z 499.25,A -85,B 0,C 180,E1 -30258.885,E2 -30258.885} C_VEL
LIN {X 0,Y 45.124,Z 511.675,A -85,B 0,C 180,E1 -30270.415,E2 -30270.415} C_VEL
LIN {X 0,Y 51.489,Z 522.699,A -85,B 0,C 180,E1 -30280.422,E2 -30280.422} C_VEL
LIN {X 0,Y 52.701,Z 524.373,A -85,B 0,C 180,E1 -30281.824,E2 -30281.824} C_VEL
LIN {X 0,Y 53.655,Z 525.767,A -85,B 0,C 180,E1 -30284.727,E2 -30284.727} C_VEL
LIN {X 0,Y 49.984,Z 518.843,A -85,B 0,C 180,E1 -30300.055,E2 -30300.055} C_VEL
LIN {X 0,Y 50.381,Z 512.06,A -85,B 0,C 180,E1 -30313.798,E2 -30313.798} C_VEL
LIN {X 0,Y 51.974,Z 506.449,A -85,B 0,C 180,E1 -30322.227,E2 -30322.227} C_VEL
LIN {X 0,Y 55.007,Z 500.444,A -85,B 0,C 180,E1 -30329.999,E2 -30329.999} C_VEL
LIN {X 0,Y 58.567,Z 496.233,A -85,B 0,C 180,E1 -30334.99,E2 -30334.99} C_VEL
LIN {X 0,Y 60.247,Z 494.856,A -85,B 0,C 180,E1 -30336.814,E2 -30336.814} C_VEL
LIN {X 0,Y 57.565,Z 499.754,A -85,B 0,C 180,E1 -30344.132,E2 -30344.132} C_VEL
LIN {X 0,Y 56.227,Z 506.847,A -85,B 0,C 180,E1 -30355.946,E2 -30355.946} C_VEL
LIN {X 0,Y 58.139,Z 513.756,A -85,B 0,C 180,E1 -30369.823,E2 -30369.823} C_VEL
LIN {X 0,Y 57.272,Z 512.439,A -85,B 0,C 180,E1 -30372.58,E2 -30372.58} C_VEL
LIN {X 0,Y 51.322,Z 501.201,A -85,B 0,C 180,E1 -30380.698,E2 -30380.698} C_VEL
LIN {X 0,Y 47.524,Z 490.471,A -85,B 0,C 180,E1 -30388.824,E2 -30388.824} C_VEL
LIN {X 0,Y 45.066,Z 480.145,A -85,B 0,C 180,E1 -30395.83,E2 -30395.83} C_VEL
LIN {X 0,Y 42.969,Z 465.679,A -85,B 0,C 180,E1 -30403.974,E2 -30403.974} C_VEL
LIN {X 0,Y 41.529,Z 448.764,A -85,B 0,C 180,E1 -30411.48,E2 -30411.48} C_VEL
LIN {X 0,Y 39.421,Z 424.46,A -85,B 0,C 180,E1 -30420.953,E2 -30420.953} C_VEL
LIN {X 0,Y 37.574,Z 398.128,A -85,B 0,C 180,E1 -30431.181,E2 -30431.181} C_VEL
LIN {X 0,Y 32.318,Z 378.152,A -85,B 0,C 180,E1 -30436.095,E2 -30436.095} C_VEL
LIN {X 0,Y 32.145,Z 377.427,A -85,B 0,C 180,E1 -30436.512,E2 -30436.512} C_VEL
LIN {X 0,Y 30.456,Z 377.582,A -85,B 0,C 180,E1 -30447.478,E2 -30447.478} C_VEL
LIN {X 0,Y 29.59,Z 377.663,A -85,B 0,C 180,E1 -30465.433,E2 -30465.433} C_VEL
LIN {X 0,Y 29.507,Z 377.672,A -85,B 0,C 180,E1 -30481.554,E2 -30481.554} C_VEL
LIN {X 0,Y 29.887,Z 377.637,A -85,B 0,C 180,E1 -30490.137,E2 -30490.137} C_VEL
LIN {X 0,Y 30.124,Z 377.616,A -85,B 0,C 180,E1 -30496.511,E2 -30496.511} C_VEL
LIN {X 0,Y 30.833,Z 377.545,A -85,B 0,C 180,E1 -30510.002,E2 -30510.002} C_VEL
LIN {X 0,Y 30.125,Z 377.615,A -85,B 0,C 180,E1 -30523.494,E2 -30523.494} C_VEL
LIN {X 0,Y 29.886,Z 377.637,A -85,B 0,C 180,E1 -30529.861,E2 -30529.861} C_VEL
LIN {X 0,Y 29.598,Z 377.657,A -85,B 0,C 180,E1 -30535.264,E2 -30535.264} C_VEL
LIN {X 0,Y 29.312,Z 378.486,A -85,B 0,C 180,E1 -30542.221,E2 -30542.221} C_VEL
LIN {X 0,Y 28.981,Z 380.448,A -85,B 0,C 180,E1 -30548.463,E2 -30548.463} C_VEL
LIN {X 0,Y 28.664,Z 383.169,A -85,B 0,C 180,E1 -30553.997,E2 -30553.997} C_VEL
LIN {X 0,Y 28.288,Z 388.18,A -85,B 0,C 180,E1 -30560.795,E2 -30560.795} C_VEL
LIN {X 0,Y 28.322,Z 396.045,A -85,B 0,C 180,E1 -30567.766,E2 -30567.766} C_VEL
LIN {X 0,Y 29.369,Z 402.167,A -85,B 0,C 180,E1 -30570.889,E2 -30570.889} C_VEL
LIN {X 0,Y 30.126,Z 405.219,A -85,B 0,C 180,E1 -30571.945,E2 -30571.945} C_VEL
LIN {X 0,Y 30.975,Z 445.449,A -85,B 0,C 180,E1 -30591.204,E2 -30591.204} C_VEL
LIN {X 0,Y 31.583,Z 463.446,A -85,B 0,C 180,E1 -30600.803,E2 -30600.803} C_VEL
LIN {X 0,Y 32.549,Z 475.972,A -85,B 0,C 180,E1 -30609.326,E2 -30609.326} C_VEL
LIN {X 0,Y 34.59,Z 488.245,A -85,B 0,C 180,E1 -30619.285,E2 -30619.285} C_VEL
LIN {X 0,Y 37.777,Z 499.344,A -85,B 0,C 180,E1 -30629.238,E2 -30629.238} C_VEL
LIN {X 0,Y 42.912,Z 510.445,A -85,B 0,C 180,E1 -30639.399,E2 -30639.399} C_VEL
LIN {X 0,Y 47.475,Z 517.681,A -85,B 0,C 180,E1 -30645.574,E2 -30645.574} C_VEL
LIN {X 0,Y 47.514,Z 517.723,A -85,B 0,C 180,E1 -30647.701,E2 -30647.701} C_VEL
LIN {X 0,Y 45.401,Z 510.067,A -85,B 0,C 180,E1 -30665.145,E2 -30665.145} C_VEL
LIN {X 0,Y 46.143,Z 505.358,A -85,B 0,C 180,E1 -30674.445,E2 -30674.445} C_VEL
LIN {X 0,Y 49.272,Z 496.806,A -85,B 0,C 180,E1 -30686.877,E2 -30686.877} C_VEL
LIN {X 0,Y 53.155,Z 491.642,A -85,B 0,C 180,E1 -30693.671,E2 -30693.671} C_VEL
LIN {X 0,Y 56.481,Z 488.883,A -85,B 0,C 180,E1 -30697.394,E2 -30697.394} C_VEL
LIN {X 0,Y 54.102,Z 492.529,A -85,B 0,C 180,E1 -30703.347,E2 -30703.347} C_VEL
LIN {X 0,Y 52.418,Z 499.99,A -85,B 0,C 180,E1 -30715.834,E2 -30715.834} C_VEL
LIN {X 0,Y 53.409,Z 505.902,A -85,B 0,C 180,E1 -30727.853,E2 -30727.853} C_VEL
LIN {X 0,Y 52.458,Z 504.379,A -85,B 0,C 180,E1 -30729.608,E2 -30729.608} C_VEL
LIN {X 0,Y 45.883,Z 490.714,A -85,B 0,C 180,E1 -30739.379,E2 -30739.379} C_VEL
LIN {X 0,Y 42.216,Z 479.096,A -85,B 0,C 180,E1 -30747.237,E2 -30747.237} C_VEL
LIN {X 0,Y 39.323,Z 464.511,A -85,B 0,C 180,E1 -30755.582,E2 -30755.582} C_VEL
LIN {X 0,Y 37.038,Z 446.914,A -85,B 0,C 180,E1 -30763.853,E2 -30763.853} C_VEL
LIN {X 0,Y 34.108,Z 423.576,A -85,B 0,C 180,E1 -30773.71,E2 -30773.71} C_VEL
LIN {X 0,Y 31.568,Z 398.577,A -85,B 0,C 180,E1 -30784.716,E2 -30784.716} C_VEL
LIN {X 0,Y 26.02,Z 378.237,A -85,B 0,C 180,E1 -30789.615,E2 -30789.615} C_VEL
LIN {X 0,Y 25.753,Z 377.974,A -85,B 0,C 180,E1 -30790.54,E2 -30790.54} C_VEL
LIN {X 0,Y 22.493,Z 378.075,A -85,B 0,C 180,E1 -30818.663,E2 -30818.663} C_VEL
LIN {X 0,Y 22.22,Z 378.084,A -85,B 0,C 180,E1 -30830.763,E2 -30830.763} C_VEL
LIN {X 0,Y 22.839,Z 378.064,A -85,B 0,C 180,E1 -30852.081,E2 -30852.081} C_VEL
LIN {X 0,Y 23.602,Z 378.041,A -85,B 0,C 180,E1 -30870.003,E2 -30870.003} C_VEL
LIN {X 0,Y 22.838,Z 378.064,A -85,B 0,C 180,E1 -30887.926,E2 -30887.926} C_VEL
LIN {X 0,Y 23.052,Z 378.058,A -85,B 0,C 180,E1 -30918.436,E2 -30918.436} C_VEL
LIN {X 0,Y 23.199,Z 378.167,A -85,B 0,C 180,E1 -30920.544,E2 -30920.544} C_VEL
LIN {X 0,Y 29.369,Z 402.167,A -85,B 0,C 180,E1 -30930.889,E2 -30930.889} C_VEL
LIN {X 0,Y 29.852,Z 405.919,A -85,B 0,C 180,E1 -30932.411,E2 -30932.411} C_VEL
LIN {X 0,Y 29.495,Z 409.654,A -85,B 0,C 180,E1 -30934.389,E2 -30934.389} C_VEL
LIN {X 0,Y 27.422,Z 416.868,A -85,B 0,C 180,E1 -30939.631,E2 -30939.631} C_VEL
LIN {X 0,Y 24.738,Z 425.955,A -85,B 0,C 180,E1 -30948.198,E2 -30948.198} C_VEL
LIN {X 0,Y 24.452,Z 431.71,A -85,B 0,C 180,E1 -30952.692,E2 -30952.692} C_VEL
LIN {X 0,Y 26.119,Z 452.366,A -85,B 0,C 180,E1 -30964.831,E2 -30964.831} C_VEL
LIN {X 0,Y 27.641,Z 468.696,A -85,B 0,C 180,E1 -30975.68,E2 -30975.68} C_VEL
LIN {X 0,Y 29.665,Z 480.014,A -85,B 0,C 180,E1 -30984.501,E2 -30984.501} C_VEL
LIN {X 0,Y 33.013,Z 491.261,A -85,B 0,C 180,E1 -30993.982,E2 -30993.982} C_VEL
LIN {X 0,Y 38.064,Z 502.537,A -85,B 0,C 180,E1 -31003.826,E2 -31003.826} C_VEL
LIN {X 0,Y 42.217,Z 509.573,A -85,B 0,C 180,E1 -31009.449,E2 -31009.449} C_VEL
LIN {X 0,Y 41.774,Z 508.213,A -85,B 0,C 180,E1 -31013.917,E2 -31013.917} C_VEL
LIN {X 0,Y 41.614,Z 500.904,A -85,B 0,C 180,E1 -31030.257,E2 -31030.257} C_VEL
LIN {X 0,Y 43.835,Z 493.079,A -85,B 0,C 180,E1 -31043.008,E2 -31043.008} C_VEL
LIN {X 0,Y 48.267,Z 486.614,A -85,B 0,C 180,E1 -31052.353,E2 -31052.353} C_VEL
LIN {X 0,Y 53.052,Z 482.686,A -85,B 0,C 180,E1 -31057.877,E2 -31057.877} C_VEL
LIN {X 0,Y 50.646,Z 485.851,A -85,B 0,C 180,E1 -31063.729,E2 -31063.729} C_VEL
LIN {X 0,Y 48.813,Z 494.306,A -85,B 0,C 180,E1 -31078.507,E2 -31078.507} C_VEL
LIN {X 0,Y 49.138,Z 497.361,A -85,B 0,C 180,E1 -31084.895,E2 -31084.895} C_VEL
LIN {X 0,Y 43.812,Z 486.749,A -85,B 0,C 180,E1 -31092.099,E2 -31092.099} C_VEL
LIN {X 0,Y 40.096,Z 476.441,A -85,B 0,C 180,E1 -31098.528,E2 -31098.528} C_VEL
LIN {X 0,Y 36.76,Z 463.105,A -85,B 0,C 180,E1 -31105.827,E2 -31105.827} C_VEL
LIN {X 0,Y 33.579,Z 445.711,A -85,B 0,C 180,E1 -31114.004,E2 -31114.004} C_VEL
LIN {X 0,Y 29.532,Z 422.085,A -85,B 0,C 180,E1 -31124.189,E2 -31124.189} C_VEL
LIN {X 0,Y 26.223,Z 398.85,A -85,B 0,C 180,E1 -31135.307,E2 -31135.307} C_VEL
LIN {X 0,Y 20.568,Z 379.34,A -85,B 0,C 180,E1 -31138.62,E2 -31138.62} C_VEL
LIN {X 0,Y 20.196,Z 378.147,A -85,B 0,C 180,E1 -31139.383,E2 -31139.383} C_VEL
LIN {X 0,Y 15.851,Z 378.178,A -85,B 0,C 180,E1 -31167.543,E2 -31167.543} C_VEL
LIN {X 0,Y 15.288,Z 378.178,A -85,B 0,C 180,E1 -31206.809,E2 -31206.809} C_VEL
LIN {X 0,Y 16.273,Z 378.178,A -85,B 0,C 180,E1 -31230.004,E2 -31230.004} C_VEL
LIN {X 0,Y 15.245,Z 378.178,A -85,B 0,C 180,E1 -31257.458,E2 -31257.458} C_VEL
LIN {X 0,Y 16.107,Z 378.178,A -85,B 0,C 180,E1 -31282.916,E2 -31282.916} C_VEL
LIN {X 0,Y 21.29,Z 398.532,A -85,B 0,C 180,E1 -31294.26,E2 -31294.26} C_VEL
LIN {X 0,Y 23.346,Z 405.336,A -85,B 0,C 180,E1 -31296.693,E2 -31296.693} C_VEL
LIN {X 0,Y 24.452,Z 431.71,A -85,B 0,C 180,E1 -31312.692,E2 -31312.692} C_VEL
LIN {X 0,Y 24.378,Z 437.324,A -85,B 0,C 180,E1 -31317.006,E2 -31317.006} C_VEL
LIN {X 0,Y 23.248,Z 446.149,A -85,B 0,C 180,E1 -31327.622,E2 -31327.622} C_VEL
LIN {X 0,Y 22.795,Z 453.139,A -85,B 0,C 180,E1 -31337.337,E2 -31337.337} C_VEL
LIN {X 0,Y 23.171,Z 458.603,A -85,B 0,C 180,E1 -31343.276,E2 -31343.276} C_VEL
LIN {X 0,Y 23.444,Z 460.489,A -85,B 0,C 180,E1 -31344.679,E2 -31344.679} C_VEL
LIN {X 0,Y 26.313,Z 474.19,A -85,B 0,C 180,E1 -31354.59,E2 -31354.59} C_VEL
LIN {X 0,Y 29.844,Z 484.955,A -85,B 0,C 180,E1 -31362.62,E2 -31362.62} C_VEL
LIN {X 0,Y 35.017,Z 496.228,A -85,B 0,C 180,E1 -31371.062,E2 -31371.062} C_VEL
LIN {X 0,Y 37.403,Z 500.408,A -85,B 0,C 180,E1 -31374.091,E2 -31374.091} C_VEL
LIN {X 0,Y 37.578,Z 500.298,A -85,B 0,C 180,E1 -31375.868,E2 -31375.868} C_VEL
LIN {X 0,Y 37.559,Z 494.83,A -85,B 0,C 180,E1 -31388.02,E2 -31388.02} C_VEL
LIN {X 0,Y 39.874,Z 486.777,A -85,B 0,C 180,E1 -31402.31,E2 -31402.31} C_VEL
LIN {X 0,Y 44.38,Z 480.607,A -85,B 0,C 180,E1 -31411.97,E2 -31411.97} C_VEL
LIN {X 0,Y 49.71,Z 476.447,A -85,B 0,C 180,E1 -31418.222,E2 -31418.222} C_VEL
LIN {X 0,Y 49.765,Z 476.458,A -85,B 0,C 180,E1 -31418.645,E2 -31418.645} C_VEL
LIN {X 0,Y 47.332,Z 479.382,A -85,B 0,C 180,E1 -31424.712,E2 -31424.712} C_VEL
LIN {X 0,Y 45.476,Z 487.794,A -85,B 0,C 180,E1 -31440.149,E2 -31440.149} C_VEL
LIN {X 0,Y 44.57,Z 486.467,A -85,B 0,C 180,E1 -31442.013,E2 -31442.013} C_VEL
LIN {X 0,Y 39.406,Z 474.547,A -85,B 0,C 180,E1 -31448.707,E2 -31448.707} C_VEL
LIN {X 0,Y 35.221,Z 460.383,A -85,B 0,C 180,E1 -31455.536,E2 -31455.536} C_VEL
LIN {X 0,Y 31.495,Z 444.853,A -85,B 0,C 180,E1 -31462.138,E2 -31462.138} C_VEL
LIN {X 0,Y 26.408,Z 421.712,A -85,B 0,C 180,E1 -31471.088,E2 -31471.088} C_VEL
LIN {X 0,Y 22.005,Z 399.116,A -85,B 0,C 180,E1 -31481.484,E2 -31481.484} C_VEL
LIN {X 0,Y 16.345,Z 379.875,A -85,B 0,C 180,E1 -31480.791,E2 -31480.791} C_VEL
LIN {X 0,Y 15.887,Z 378.178,A -85,B 0,C 180,E1 -31481.216,E2 -31481.216} C_VEL
LIN {X 0,Y 10.867,Z 378.178,A -85,B 0,C 180,E1 -31499.982,E2 -31499.982} C_VEL
LIN {X 0,Y 8.103,Z 378.178,A -85,B 0,C 180,E1 -31529.867,E2 -31529.867} C_VEL
LIN {X 0,Y 7.879,Z 378.178,A -85,B 0,C 180,E1 -31563.075,E2 -31563.075} C_VEL
LIN {X 0,Y 8.707,Z 378.178,A -85,B 0,C 180,E1 -31590.008,E2 -31590.008} C_VEL
LIN {X 0,Y 8.122,Z 378.178,A -85,B 0,C 180,E1 -31620.128,E2 -31620.128} C_VEL
LIN {X 0,Y 9.046,Z 378.178,A -85,B 0,C 180,E1 -31649.549,E2 -31649.549} C_VEL
LIN {X 0,Y 14.022,Z 396.342,A -85,B 0,C 180,E1 -31662.852,E2 -31662.852} C_VEL
LIN {X 0,Y 16.971,Z 405.703,A -85,B 0,C 180,E1 -31666.085,E2 -31666.085} C_VEL
LIN {X 0,Y 20.934,Z 443.36,A -85,B 0,C 180,E1 -31693.354,E2 -31693.354} C_VEL
LIN {X 0,Y 23.444,Z 460.489,A -85,B 0,C 180,E1 -31704.679,E2 -31704.679} C_VEL
LIN {X 0,Y 24.237,Z 465.927,A -85,B 0,C 180,E1 -31709.81,E2 -31709.81} C_VEL
LIN {X 0,Y 25.1,Z 470.946,A -85,B 0,C 180,E1 -31716.919,E2 -31716.919} C_VEL
LIN {X 0,Y 29.852,Z 483.549,A -85,B 0,C 180,E1 -31735.276,E2 -31735.276} C_VEL
LIN {X 0,Y 31.558,Z 486.879,A -85,B 0,C 180,E1 -31737.986,E2 -31737.986} C_VEL
LIN {X 0,Y 33.514,Z 490.503,A -85,B 0,C 180,E1 -31740.12,E2 -31740.12} C_VEL
LIN {X 0,Y 33.737,Z 489.77,A -85,B 0,C 180,E1 -31742.789,E2 -31742.789} C_VEL
LIN {X 0,Y 35.733,Z 481.247,A -85,B 0,C 180,E1 -31759.579,E2 -31759.579} C_VEL
LIN {X 0,Y 40.285,Z 474.9,A -85,B 0,C 180,E1 -31770.712,E2 -31770.712} C_VEL
LIN {X 0,Y 46.004,Z 470.387,A -85,B 0,C 180,E1 -31777.916,E2 -31777.916} C_VEL
LIN {X 0,Y 47.048,Z 469.878,A -85,B 0,C 180,E1 -31779.009,E2 -31779.009} C_VEL
LIN {X 0,Y 43.666,Z 474.006,A -85,B 0,C 180,E1 -31788.311,E2 -31788.311} C_VEL
LIN {X 0,Y 42.885,Z 476.24,A -85,B 0,C 180,E1 -31792.7,E2 -31792.7} C_VEL
LIN {X 0,Y 42.269,Z 477.584,A -85,B 0,C 180,E1 -31796.607,E2 -31796.607} C_VEL
LIN {X 0,Y 38.685,Z 468.968,A -85,B 0,C 180,E1 -31800.341,E2 -31800.341} C_VEL
LIN {X 0,Y 34.62,Z 456.435,A -85,B 0,C 180,E1 -31805.07,E2 -31805.07} C_VEL
LIN {X 0,Y 30.729,Z 442.903,A -85,B 0,C 180,E1 -31809.467,E2 -31809.467} C_VEL
LIN {X 0,Y 25.08,Z 421.343,A -85,B 0,C 180,E1 -31815.519,E2 -31815.519} C_VEL
LIN {X 0,Y 19.648,Z 399.222,A -85,B 0,C 180,E1 -31822.716,E2 -31822.716} C_VEL
LIN {X 0,Y 14.611,Z 380.22,A -85,B 0,C 180,E1 -31815.136,E2 -31815.136} C_VEL
LIN {X 0,Y 14.056,Z 378.178,A -85,B 0,C 180,E1 -31814.715,E2 -31814.715} C_VEL
LIN {X 0,Y 9.583,Z 378.178,A -85,B 0,C 180,E1 -31817.163,E2 -31817.163} C_VEL
LIN {X 0,Y 0.756,Z 378.178,A -85,B 0,C 180,E1 -31950.09,E2 -31950.09} C_VEL
LIN {X 0,Y 2.908,Z 378.178,A -85,B 0,C 180,E1 -32052.445,E2 -32052.445} C_VEL
LIN {X 0,Y 8.197,Z 395.716,A -85,B 0,C 180,E1 -32047.471,E2 -32047.471} C_VEL
LIN {X 0,Y 11.474,Z 405.877,A -85,B 0,C 180,E1 -32045.489,E2 -32045.489} C_VEL
LIN {X 0,Y 17.511,Z 439.233,A -85,B 0,C 180,E1 -32070.721,E2 -32070.721} C_VEL
LIN {X 0,Y 21.048,Z 455.262,A -85,B 0,C 180,E1 -32079.737,E2 -32079.737} C_VEL
LIN {X 0,Y 25.137,Z 470.924,A -85,B 0,C 180,E1 -32088.722,E2 -32088.722} C_VEL
LIN {X 0,Y 29.756,Z 483.036,A -85,B 0,C 180,E1 -32095.767,E2 -32095.767} C_VEL
LIN {X 0,Y 31.558,Z 486.879,A -85,B 0,C 180,E1 -32097.986,E2 -32097.986} C_VEL
LIN {X 0,Y 31.555,Z 486.267,A -85,B 0,C 180,E1 -32099.534,E2 -32099.534} C_VEL
LIN {X 0,Y 30.23,Z 481.941,A -85,B 0,C 180,E1 -32101.846,E2 -32101.846} C_VEL
LIN {X 0,Y 25.931,Z 468.672,A -85,B 0,C 180,E1 -32102.684,E2 -32102.684} C_VEL
LIN {X 0,Y 22.289,Z 456.567,A -85,B 0,C 180,E1 -32099.382,E2 -32099.382} C_VEL
LIN {X 0,Y 18.04,Z 441.308,A -85,B 0,C 180,E1 -32094.673,E2 -32094.673} C_VEL
LIN {X 0,Y 9.271,Z 406.456,A -85,B 0,C 180,E1 -32083.952,E2 -32083.952} C_VEL
LIN {X 0,Y 6.364,Z 383.627,A -85,B 0,C 180,E1 -32135.336,E2 -32135.336} C_VEL
LIN {X 0,Y 10.677,Z 383.6,A -85,B 0,C 180,E1 -32151.324,E2 -32151.324} C_VEL
LIN {X 0,Y 13.735,Z 387.358,A -85,B 0,C 180,E1 -32151.922,E2 -32151.922} C_VEL
LIN {X 0,Y 16.15,Z 388.831,A -85,B 0,C 180,E1 -32153.495,E2 -32153.495} C_VEL
LIN {X 0,Y 17.846,Z 389.129,A -85,B 0,C 180,E1 -32155.12,E2 -32155.12} C_VEL
LIN {X 0,Y 20.218,Z 400.686,A -85,B 0,C 180,E1 -32162.062,E2 -32162.062} C_VEL
LIN {X 0,Y 29.038,Z 432.198,A -85,B 0,C 180,E1 -32158.143,E2 -32158.143} C_VEL
LIN {X 0,Y 33.865,Z 448.213,A -85,B 0,C 180,E1 -32155.636,E2 -32155.636} C_VEL
LIN {X 0,Y 38.673,Z 462.21,A -85,B 0,C 180,E1 -32152.203,E2 -32152.203} C_VEL
LIN {X 0,Y 40.785,Z 467.593,A -85,B 0,C 180,E1 -32150.497,E2 -32150.497} C_VEL
LIN {X 0,Y 44.065,Z 463.506,A -85,B 0,C 180,E1 -32140.388,E2 -32140.388} C_VEL
LIN {X 0,Y 44.521,Z 463.253,A -85,B 0,C 180,E1 -32139.381,E2 -32139.381} C_VEL
LIN {X 0,Y 39.449,Z 466.321,A -85,B 0,C 180,E1 -32133.88,E2 -32133.88} C_VEL
LIN {X 0,Y 33.837,Z 472.094,A -85,B 0,C 180,E1 -32123.209,E2 -32123.209} C_VEL
LIN {X 0,Y 31.005,Z 477.957,A -85,B 0,C 180,E1 -32111.022,E2 -32111.022} C_VEL
LIN {X 0,Y 30.433,Z 479.051,A -85,B 0,C 180,E1 -32107.493,E2 -32107.493} C_VEL
LIN {X 0,Y 25.25,Z 466.21,A -85,B 0,C 180,E1 -32102.818,E2 -32102.818} C_VEL
LIN {X 0,Y 22.289,Z 456.567,A -85,B 0,C 180,E1 -32099.382,E2 -32099.382} C_VEL
LIN {X 0,Y 20.809,Z 450.867,A -85,B 0,C 180,E1 -32099.068,E2 -32099.068} C_VEL
LIN {X 0,Y 19.687,Z 445.121,A -85,B 0,C 180,E1 -32102.092,E2 -32102.092} C_VEL
LIN {X 0,Y 17.848,Z 431.728,A -85,B 0,C 180,E1 -32113.525,E2 -32113.525} C_VEL
LIN {X 0,Y 16.663,Z 425.921,A -85,B 0,C 180,E1 -32115.981,E2 -32115.981} C_VEL
LIN {X 0,Y 11.901,Z 406.356,A -85,B 0,C 180,E1 -32121.59,E2 -32121.59} C_VEL
LIN {X 0,Y 12.093,Z 394.15,A -85,B 0,C 180,E1 -32140.869,E2 -32140.869} C_VEL
LIN {X 0,Y 13.221,Z 395.047,A -85,B 0,C 180,E1 -32142.562,E2 -32142.562} C_VEL
LIN {X 0,Y 23.125,Z 413.909,A -85,B 0,C 180,E1 -32142.947,E2 -32142.947} C_VEL
LIN {X 0,Y 25.574,Z 417.182,A -85,B 0,C 180,E1 -32143.835,E2 -32143.835} C_VEL
LIN {X 0,Y 27.226,Z 418.285,A -85,B 0,C 180,E1 -32144.957,E2 -32144.957} C_VEL
LIN {X 0,Y 27.754,Z 418.267,A -85,B 0,C 180,E1 -32145.486,E2 -32145.486} C_VEL
LIN {X 0,Y 32.994,Z 435.698,A -85,B 0,C 180,E1 -32145.681,E2 -32145.681} C_VEL
LIN {X 0,Y 37.228,Z 448.797,A -85,B 0,C 180,E1 -32144.953,E2 -32144.953} C_VEL
LIN {X 0,Y 40.408,Z 457.538,A -85,B 0,C 180,E1 -32143.761,E2 -32143.761} C_VEL
LIN {X 0,Y 41.143,Z 457.161,A -85,B 0,C 180,E1 -32142.006,E2 -32142.006} C_VEL
LIN {X 0,Y 41.983,Z 456.644,A -85,B 0,C 180,E1 -32139.939,E2 -32139.939} C_VEL
LIN {X 0,Y 36.559,Z 459.701,A -85,B 0,C 180,E1 -32133.793,E2 -32133.793} C_VEL
LIN {X 0,Y 30.622,Z 465.7,A -85,B 0,C 180,E1 -32121.257,E2 -32121.257} C_VEL
LIN {X 0,Y 29.394,Z 467.628,A -85,B 0,C 180,E1 -32116.825,E2 -32116.825} C_VEL
LIN {X 0,Y 24.348,Z 453.019,A -85,B 0,C 180,E1 -32114.751,E2 -32114.751} C_VEL
LIN {X 0,Y 20.062,Z 438.622,A -85,B 0,C 180,E1 -32114.483,E2 -32114.483} C_VEL
LIN {X 0,Y 16.663,Z 425.921,A -85,B 0,C 180,E1 -32115.981,E2 -32115.981} C_VEL
LIN {X 0,Y 17.038,Z 425.525,A -85,B 0,C 180,E1 -32118.308,E2 -32118.308} C_VEL
LIN {X 0,Y 18.616,Z 426.39,A -85,B 0,C 180,E1 -32123.26,E2 -32123.26} C_VEL
LIN {X 0,Y 22.172,Z 430.226,A -85,B 0,C 180,E1 -32129.327,E2 -32129.327} C_VEL
LIN {X 0,Y 28.849,Z 440.362,A -85,B 0,C 180,E1 -32134.272,E2 -32134.272} C_VEL
LIN {X 0,Y 32.818,Z 447.958,A -85,B 0,C 180,E1 -32135.301,E2 -32135.301} C_VEL
LIN {X 0,Y 33.895,Z 450.61,A -85,B 0,C 180,E1 -32135.188,E2 -32135.188} C_VEL
LIN {X 0,Y 34.442,Z 452.599,A -85,B 0,C 180,E1 -32134.827,E2 -32134.827} C_VEL
LIN {X 0,Y 30.841,Z 455.456,A -85,B 0,C 180,E1 -32128.326,E2 -32128.326} C_VEL
LIN {X 0,Y 29.878,Z 455.582,A -85,B 0,C 180,E1 -32126.546,E2 -32126.546} C_VEL
LIN {X 0,Y 25.27,Z 440.465,A -85,B 0,C 180,E1 -32127.979,E2 -32127.979} C_VEL
LIN {X 0,Y 20.397,Z 420.582,A -85,B 0,C 180,E1 -32133.464,E2 -32133.464} C_VEL
LIN {X 0,Y 23.316,Z 423.539,A -85,B 0,C 180,E1 -32136.644,E2 -32136.644} C_VEL
LIN {X 0,Y 33.895,Z 450.61,A -85,B 0,C 180,E1 -32135.188,E2 -32135.188} C_VEL
LIN {X 0,Y 34.021,Z 451.313,A -85,B 0,C 180,E1 -32135.162,E2 -32135.162} C_VEL
LIN {X 0,Y 34.021,Z 600,A -85,B 0,C 180,E1 -32135.162,E2 -32135.162} C_VEL
LIN {X 0,Y 34.021,Z 600,A -85,B 0,C 180,E1 -32135.162,E2 -32135.162}

QRS_NEXT_CUT()

QRS_NEXT()
QRS_HOME()

END
